// TwinCAT 3 PLC project OSCAT
// Title: OSCAT
// Company: RWTH Aachen University - E.ON Energy Research Center
// ProjectVersion: 1.1.2
// Description: This library is based on the OSCAT library (http://www.oscat.de/)
// ProgramVersion: 3.1.4022.1
// libraries:
//   Tc2_Standard, * (Beckhoff Automation GmbH)
// project tree:
//   oscat_basic/Data types/ CALENDAR.TcDUT (not stored), COMPLEX.TcDUT, CONSTANTS_LANGUAGE.TcDUT (not stored), CONSTANTS_LOCATION.TcDUT, CONSTANTS_MATH.TcDUT, CONSTANTS_PHYS.TcDUT, CONSTANTS_SETUP.TcDUT, ESR_DATA.TcDUT (not stored), CONTROL_MODE.TcDUT, FRACTION.TcDUT, HOLIDAY_DATA.TcDUT (not stored), REAL2.TcDUT, SDT.TcDUT, CONTROL_PARAMETERS.TcDUT, IO_TERMINAL_PARAMETERS.TcDUT, TIMER_EVENT.TcDUT (not stored), VECTOR_3.TcDUT
//   oscat_basic/Global Variables/ Constants_2.TcGVL, Globale_Variablen_2.TcGVL (not stored)
//   oscat_basic/POUs/Buffer Management/ BUFFER_COMP.TcPOU (not stored), BUFFER_SEARCH.TcPOU, BUFFER_TO_STRING.TcPOU, _BUFFER_INSERT.TcPOU, _BUFFER_UPPERCASE.TcPOU, _STRING_TO_BUFFER.TcPOU (not stored)
//   oscat_basic/POUs/Engineering/automation/ DRIVER_1.TcPOU, DRIVER_4.TcPOU (not stored), DRIVER_4C.TcPOU (not stored), FLOW_CONTROL.TcPOU, FT_Profile.TcPOU (not stored), INC_DEC.TcPOU (not stored), INTERLOCK.TcPOU, INTERLOCK_4.TcPOU, MANUAL.TcPOU, MANUAL_1.TcPOU, MANUAL_2.TcPOU (not stored), MANUAL_4.TcPOU (not stored), PARSET.TcPOU (not stored), PARSET2.TcPOU, SIGNAL.TcPOU (not stored), SIGNAL_4.TcPOU, SRAMP.TcPOU (not stored), TUNE.TcPOU (not stored), TUNE2.TcPOU (not stored)
//   oscat_basic/POUs/Engineering/Control/ BAND_B.TcPOU (not stored), CONTROL_SET1.TcPOU, CONTROL_SET2.TcPOU, CTRL_IN.TcPOU, CTRL_OUT.TcPOU, CTRL_PI.TcPOU, CTRL_PID.TcPOU, CTRL_PWM.TcPOU (not stored), DEAD_BAND.TcPOU (not stored), DEAD_BAND_A.TcPOU, DEAD_ZONE.TcPOU (not stored), DEAD_ZONE2.TcPOU (not stored), VOLTAGE_CONTROL.TcPOU, FB_CONTROL.TcPOU, FB_Integrate.TcPOU, FB_PID.TcPOU, FT_DERIV.TcPOU (not stored), FT_IMP.TcPOU, FT_INT.TcPOU (not stored), FT_INT2.TcPOU (not stored), FT_PD.TcPOU (not stored), FT_PDT1.TcPOU (not stored), FT_PI.TcPOU, FT_PID.TcPOU, FT_PIDW.TcPOU (not stored), FT_PIDWL.TcPOU, FT_PIW.TcPOU, FT_PIWL.TcPOU (not stored), FT_PT1.TcPOU, FT_PT2.TcPOU (not stored), FT_TN16.TcPOU, FT_TN64.TcPOU, FT_TN8.TcPOU, HYST.TcPOU, HYST_1.TcPOU, HYST_2.TcPOU, HYST_3.TcPOU, INTEGRATE.TcPOU (not stored)
//   oscat_basic/POUs/Engineering/Conversion/ ASTRO.TcPOU (not stored), BFT_TO_MS.TcPOU (not stored), C_TO_F.TcPOU, C_TO_K.TcPOU, DEG_TO_DIR.TcPOU, DIR_TO_DEG.TcPOU (not stored), ENERGY.TcPOU, F_TO_C.TcPOU (not stored), F_TO_OM.TcPOU (not stored), F_TO_PT.TcPOU, GEO_TO_DEG.TcPOU (not stored), KMH_TO_MS.TcPOU, K_TO_C.TcPOU (not stored), LENGTH.TcPOU (not stored), MS_TO_BFT.TcPOU (not stored), MS_TO_KMH.TcPOU, OM_TO_F.TcPOU (not stored), PRESSURE.TcPOU (not stored), PT_TO_F.TcPOU (not stored), SPEED.TcPOU (not stored), TEMPERATURE.TcPOU (not stored)
//   oscat_basic/POUs/Engineering/measurements/ ALARM_2.TcPOU (not stored), BAR_GRAPH.TcPOU (not stored), CALIBRATE.TcPOU, CYCLE_TIME.TcPOU (not stored), DT_SIMU.TcPOU (not stored), FLOW_METER.TcPOU, METER.TcPOU (not stored), METER_STAT.TcPOU, M_D.TcPOU, M_T.TcPOU (not stored), M_TX.TcPOU (not stored), ONTIME.TcPOU (not stored), TC_MS.TcPOU, TC_S.TcPOU (not stored), TC_US.TcPOU (not stored), T_PLC_MS.TcPOU (not stored), T_PLC_US.TcPOU
//   oscat_basic/POUs/Engineering/sensor/ MULTI_IN.TcPOU (not stored), RES_NI.TcPOU (not stored), RES_NTC.TcPOU, RES_PT.TcPOU, RES_SI.TcPOU (not stored), SENSOR_INT.TcPOU (not stored), TEMP_NI.TcPOU (not stored), TEMP_NTC.TcPOU, TEMP_PT.TcPOU, TEMP_SI.TcPOU
//   oscat_basic/POUs/Engineering/signal generators/ GEN_PULSE.TcPOU, GEN_PW2.TcPOU, GEN_RDM.TcPOU (not stored), GEN_RDT.TcPOU (not stored), GEN_RMP.TcPOU (not stored), GEN_SIN.TcPOU (not stored), GEN_SQR.TcPOU, PWM_DC.TcPOU (not stored), PWM_PW.TcPOU (not stored), RMP_B.TcPOU, RMP_SOFT.TcPOU, RMP_W.TcPOU, _RMP_B.TcPOU, _RMP_NEXT.TcPOU (not stored), _RMP_W.TcPOU (not stored)
//   oscat_basic/POUs/Engineering/signal processing/ AIN.TcPOU (not stored), AIN1.TcPOU, AOUT.TcPOU, AOUT1.TcPOU, BYTE_TO_RANGE.TcPOU, DELAY.TcPOU, DELAY_200.TcPOU, DELAY_4.TcPOU (not stored), FADE.TcPOU, FB_InLinear.TcPOU, FB_InOnOff.TcPOU, FB_OutLinear.TcPOU, FB_OutOnOff.TcPOU, FILTER_DW.TcPOU, FILTER_I.TcPOU, FILTER_MAV_DW.TcPOU (not stored), FILTER_MAV_W.TcPOU, FILTER_W.TcPOU (not stored), FILTER_WAV.TcPOU (not stored), MIX.TcPOU (not stored), MUX_R2.TcPOU (not stored), MUX_R4.TcPOU (not stored), OFFSET.TcPOU (not stored), OFFSET2.TcPOU (not stored), OVERRIDE.TcPOU, RANGE_TO_BYTE.TcPOU, RANGE_TO_WORD.TcPOU, SCALE.TcPOU (not stored), SCALE_B.TcPOU, SCALE_B2.TcPOU, SCALE_B4.TcPOU, SCALE_B8.TcPOU (not stored), SCALE_D.TcPOU, SCALE_R.TcPOU, SCALE_X2.TcPOU (not stored), SCALE_X4.TcPOU (not stored), SCALE_X8.TcPOU (not stored), SEL2_OF_3.TcPOU, SEL2_OF_3B.TcPOU (not stored), SH.TcPOU (not stored), SH_1.TcPOU, SH_2.TcPOU, SH_T.TcPOU, STAIR.TcPOU (not stored), STAIR2.TcPOU (not stored), TREND.TcPOU, TREND_DW.TcPOU (not stored), WORD_TO_RANGE.TcPOU
//   oscat_basic/POUs/List Processing/ LIST_ADD.TcPOU (not stored), LIST_CLEAN.TcPOU (not stored), LIST_GET.TcPOU, LIST_INSERT.TcPOU (not stored), LIST_LEN.TcPOU, LIST_NEXT.TcPOU, LIST_RETRIEVE.TcPOU (not stored), LIST_RETRIEVE_LAST.TcPOU (not stored)
//   oscat_basic/POUs/Logic/FF edge triggered/ COUNT_BR.TcPOU, COUNT_DR.TcPOU (not stored), FF_D2E.TcPOU, FF_D4E.TcPOU (not stored), FF_DRE.TcPOU, FF_JKE.TcPOU, FF_RSE.TcPOU (not stored), SELECT_8.TcPOU, SHR_4E.TcPOU (not stored), SHR_4UDE.TcPOU, SHR_8PLE.TcPOU (not stored), SHR_8UDE.TcPOU, TOGGLE.TcPOU (not stored)
//   oscat_basic/POUs/Logic/FF pulse triggered/ LTCH.TcPOU (not stored), LTCH_4.TcPOU (not stored), STORE_8.TcPOU
//   oscat_basic/POUs/Logic/gate logic/ BCDC_TO_INT.TcPOU, BIT_COUNT.TcPOU, BIT_LOAD_B.TcPOU, BIT_LOAD_B2.TcPOU, BIT_LOAD_DW.TcPOU, BIT_LOAD_DW2.TcPOU (not stored), BIT_LOAD_W.TcPOU (not stored), BIT_LOAD_W2.TcPOU, BIT_OF_DWORD.TcPOU (not stored), BIT_TOGGLE_B.TcPOU (not stored), BIT_TOGGLE_DW.TcPOU, BIT_TOGGLE_W.TcPOU, BYTE_OF_BIT.TcPOU (not stored), BYTE_OF_DWORD.TcPOU, BYTE_TO_BITS.TcPOU (not stored), BYTE_TO_GRAY.TcPOU, CHECK_PARITY.TcPOU (not stored), CHK_REAL.TcPOU, DEC_2.TcPOU, DEC_4.TcPOU, DEC_8.TcPOU (not stored), DWORD_OF_BYTE.TcPOU (not stored), DWORD_OF_WORD.TcPOU, DW_TO_REAL.TcPOU, GRAY_TO_BYTE.TcPOU, INT_TO_BCDC.TcPOU (not stored), MUX_2.TcPOU, MUX_4.TcPOU, PARITY.TcPOU, REAL_TO_DW.TcPOU, REFLECT.TcPOU, REVERSE.TcPOU (not stored), SHL1.TcPOU, SHR1.TcPOU (not stored), SWAP_BYTE.TcPOU (not stored), SWAP_BYTE2.TcPOU (not stored), WORD_OF_BYTE.TcPOU (not stored), WORD_OF_DWORD.TcPOU
//   oscat_basic/POUs/Logic/generators/ A_TRIG.TcPOU (not stored), B_TRIG.TcPOU, CLICK_CNT.TcPOU, CLICK_DEC.TcPOU (not stored), CLK_DIV.TcPOU (not stored), CLK_N.TcPOU (not stored), CLK_PRG.TcPOU, CLK_PULSE.TcPOU, CYCLE_4.TcPOU (not stored), D_TRIG.TcPOU, GEN_BIT.TcPOU (not stored), GEN_SQ.TcPOU, SCHEDULER.TcPOU (not stored), SCHEDULER_2.TcPOU (not stored), SEQUENCE_4.TcPOU (not stored), SEQUENCE_64.TcPOU, SEQUENCE_8.TcPOU, TMAX.TcPOU, TMIN.TcPOU, TOF_1.TcPOU (not stored), TONOF.TcPOU, TP_1.TcPOU (not stored), TP_1D.TcPOU (not stored), TP_X.TcPOU
//   oscat_basic/POUs/Logic/memory/ FIFO_16.TcPOU (not stored), FIFO_32.TcPOU, STACK_16.TcPOU, STACK_32.TcPOU
//   oscat_basic/POUs/Logic/Others/ CRC_GEN.TcPOU (not stored), MATRIX.TcPOU (not stored), PIN_CODE.TcPOU
//   oscat_basic/POUs/Mathematical/ ACOSH.TcPOU, ACOTH.TcPOU (not stored), AGDF.TcPOU (not stored), ASINH.TcPOU, ATAN2.TcPOU (not stored), ATANH.TcPOU (not stored), BETA.TcPOU, BINOM.TcPOU, CAUCHY.TcPOU, CAUCHYCD.TcPOU (not stored), CEIL.TcPOU (not stored), CEIL2.TcPOU (not stored), CMP.TcPOU, COSH.TcPOU, COTH.TcPOU, DEC1.TcPOU, DEG.TcPOU (not stored), DIFFER.TcPOU (not stored), D_TRUNC.TcPOU, ERF.TcPOU, ERFC.TcPOU, EVEN.TcPOU, EXP10.TcPOU, EXPN.TcPOU (not stored), FACT.TcPOU (not stored), FIB.TcPOU, FLOOR.TcPOU (not stored), FLOOR2.TcPOU, FRACT.TcPOU (not stored), GAMMA.TcPOU, GAUSS.TcPOU, GAUSSCD.TcPOU, GCD.TcPOU (not stored), GDF.TcPOU, GOLD.TcPOU, HYPOT.TcPOU, INC.TcPOU (not stored), INC1.TcPOU, INC2.TcPOU (not stored), INV.TcPOU (not stored), LAMBERT_W.TcPOU (not stored), LANGEVIN.TcPOU, MAX3.TcPOU, MID3.TcPOU, MIN3.TcPOU (not stored), MODR.TcPOU, MUL_ADD.TcPOU, NEGX.TcPOU, RAD.TcPOU (not stored), RDM.TcPOU (not stored), RDM2.TcPOU, RDMDW.TcPOU, REAL_TO_FRAC.TcPOU, RND.TcPOU (not stored), ROUND.TcPOU (not stored), SGN.TcPOU, SIGMOID.TcPOU, SIGN_I.TcPOU (not stored), SIGN_R.TcPOU (not stored), SINC.TcPOU, SINH.TcPOU (not stored), SQRTN.TcPOU, TANC.TcPOU, TANH.TcPOU, WINDOW.TcPOU, WINDOW2.TcPOU
//   oscat_basic/POUs/Mathematical/Array/ ARRAY_AVG.TcPOU (not stored), ARRAY_GAV.TcPOU, ARRAY_HAV.TcPOU, ARRAY_MAX.TcPOU, ARRAY_MIN.TcPOU (not stored), ARRAY_SDV.TcPOU (not stored), ARRAY_SPR.TcPOU, ARRAY_SUM.TcPOU, ARRAY_TREND.TcPOU (not stored), ARRAY_VAR.TcPOU (not stored), IS_SORTED.TcPOU (not stored), _ARRAY_ABS.TcPOU (not stored), _ARRAY_ADD.TcPOU (not stored), _ARRAY_INIT.TcPOU (not stored), _ARRAY_MEDIAN.TcPOU (not stored), _ARRAY_MUL.TcPOU (not stored), _ARRAY_SHUFFLE.TcPOU (not stored), _ARRAY_SORT.TcPOU (not stored)
//   oscat_basic/POUs/Mathematical/Complex/ CABS.TcPOU (not stored), CACOS.TcPOU (not stored), CACOSH.TcPOU (not stored), CADD.TcPOU (not stored), CARG.TcPOU (not stored), CASIN.TcPOU (not stored), CASINH.TcPOU (not stored), CATAN.TcPOU (not stored), CATANH.TcPOU (not stored), CCON.TcPOU (not stored), CCOS.TcPOU (not stored), CCOSH.TcPOU (not stored), CDIV.TcPOU (not stored), CEXP.TcPOU (not stored), CINV.TcPOU (not stored), CLOG.TcPOU (not stored), CMUL.TcPOU (not stored), CPOL.TcPOU (not stored), CPOW.TcPOU (not stored), CSET.TcPOU (not stored), CSIN.TcPOU (not stored), CSINH.TcPOU (not stored), CSQRT.TcPOU (not stored), CSUB.TcPOU (not stored), CTAN.TcPOU (not stored), CTANH.TcPOU (not stored)
//   oscat_basic/POUs/Mathematical/Double Precision/ R2_ABS.TcPOU (not stored), R2_ADD.TcPOU (not stored), R2_ADD2.TcPOU (not stored), R2_MUL.TcPOU (not stored), R2_SET.TcPOU (not stored)
//   oscat_basic/POUs/Mathematical/functions/ FRMP_B.TcPOU (not stored), FT_AVG.TcPOU (not stored), FT_AVG_200.TcPOU (not stored), FT_MIN_MAX.TcPOU (not stored), FT_RMP.TcPOU (not stored), F_LIN.TcPOU (not stored), F_LIN2.TcPOU (not stored), F_POLY.TcPOU (not stored), F_POWER.TcPOU (not stored), F_QUAD.TcPOU (not stored), LINEAR_INT.TcPOU (not stored), POLYNOM_INT.TcPOU (not stored)
//   oscat_basic/POUs/Mathematical/Geometry/ CIRCLE_A.TcPOU (not stored), CIRCLE_C.TcPOU (not stored), CIRCLE_SEG.TcPOU (not stored), CONE_V.TcPOU (not stored), ELLIPSE_A.TcPOU (not stored), ELLIPSE_C.TcPOU (not stored), SPHERE_V.TcPOU (not stored), TRIANGLE_A.TcPOU (not stored)
//   oscat_basic/POUs/Mathematical/Vektormathematik/ V3_ABS.TcPOU (not stored), V3_ADD.TcPOU (not stored), V3_ANG.TcPOU (not stored), V3_DPRO.TcPOU (not stored), V3_NORM.TcPOU (not stored), V3_NUL.TcPOU (not stored), V3_PAR.TcPOU (not stored), V3_REV.TcPOU (not stored), V3_SMUL.TcPOU (not stored), V3_SUB.TcPOU (not stored), V3_XANG.TcPOU (not stored), V3_XPRO.TcPOU (not stored), V3_YANG.TcPOU (not stored), V3_ZANG.TcPOU (not stored)
//   oscat_basic/POUs/Other/ ESR_COLLECT.TcPOU, ESR_MON_B8.TcPOU (not stored), ESR_MON_R4.TcPOU, ESR_MON_X8.TcPOU (not stored), OSCAT_VERSION.TcPOU (not stored), STATUS_TO_ESR.TcPOU
//   oscat_basic/POUs/String/ BIN_TO_BYTE.TcPOU (not stored), BIN_TO_DWORD.TcPOU, BYTE_TO_STRB.TcPOU (not stored), BYTE_TO_STRH.TcPOU, CAPITALIZE.TcPOU, CHARCODE.TcPOU, CHARNAME.TcPOU, CHR_TO_STRING.TcPOU (not stored), CLEAN.TcPOU (not stored), CODE.TcPOU (not stored), COUNT_CHAR.TcPOU (not stored), COUNT_SUBSTRING.TcPOU (not stored), DEC_TO_BYTE.TcPOU (not stored), DEC_TO_DWORD.TcPOU, DEC_TO_INT.TcPOU (not stored), DEL_CHARS.TcPOU (not stored), DT_TO_STRF.TcPOU (not stored), DWORD_TO_STRB.TcPOU, DWORD_TO_STRF.TcPOU (not stored), DWORD_TO_STRH.TcPOU (not stored), EXEC.TcPOU (not stored), FILL.TcPOU (not stored), FINDB.TcPOU (not stored), FINDB_NONUM.TcPOU, FINDB_NUM.TcPOU (not stored), FINDP.TcPOU, FIND_CHAR.TcPOU, FIND_CTRL.TcPOU, FIND_NONUM.TcPOU (not stored), FIND_NUM.TcPOU (not stored), FIX.TcPOU, FLOAT_TO_REAL.TcPOU, FSTRING_TO_BYTE.TcPOU (not stored), FSTRING_TO_DT.TcPOU, FSTRING_TO_DWORD.TcPOU, FSTRING_TO_MONTH.TcPOU, FSTRING_TO_WEEK.TcPOU (not stored), FSTRING_TO_WEEKDAY.TcPOU (not stored), HEX_TO_BYTE.TcPOU, HEX_TO_DWORD.TcPOU, ISC_ALPHA.TcPOU, ISC_CTRL.TcPOU (not stored), ISC_HEX.TcPOU, ISC_LOWER.TcPOU (not stored), ISC_NUM.TcPOU (not stored), ISC_UPPER.TcPOU, IS_ALNUM.TcPOU, IS_ALPHA.TcPOU (not stored), IS_CC.TcPOU, IS_CTRL.TcPOU (not stored), IS_HEX.TcPOU, IS_LOWER.TcPOU, IS_NCC.TcPOU (not stored), IS_NUM.TcPOU, IS_UPPER.TcPOU (not stored), LOWERCASE.TcPOU (not stored), MESSAGE_4R.TcPOU, MESSAGE_8.TcPOU (not stored), MIRROR.TcPOU, MONTH_TO_STRING.TcPOU, OCT_TO_BYTE.TcPOU, OCT_TO_DWORD.TcPOU (not stored), REAL_TO_STRF.TcPOU, REPLACE_ALL.TcPOU (not stored), REPLACE_CHARS.TcPOU, REPLACE_UML.TcPOU, TICKER.TcPOU, TO_LOWER.TcPOU (not stored), TO_UML.TcPOU, TO_UPPER.TcPOU (not stored), TRIM.TcPOU, TRIM1.TcPOU (not stored), TRIME.TcPOU, UPPERCASE.TcPOU, WEEKDAY_TO_STRING.TcPOU
//   oscat_basic/POUs/Time&Date/ CALENDAR_CALC.TcPOU (not stored), DATE_ADD.TcPOU, DAYS_DELTA.TcPOU, DAYS_IN_MONTH.TcPOU, DAYS_IN_YEAR.TcPOU (not stored), DAY_OF_DATE.TcPOU (not stored), DAY_OF_MONTH.TcPOU, DAY_OF_WEEK.TcPOU (not stored), DAY_OF_YEAR.TcPOU, DAY_TO_TIME.TcPOU (not stored), DCF77.TcPOU (not stored), DST.TcPOU, DT2_TO_SDT.TcPOU (not stored), DT_TO_SDT.TcPOU, EASTER.TcPOU (not stored), EVENTS.TcPOU (not stored), HOLIDAY.TcPOU, HOUR.TcPOU (not stored), HOUR_OF_DT.TcPOU (not stored), HOUR_TO_TIME.TcPOU, HOUR_TO_TOD.TcPOU (not stored), JD2000.TcPOU (not stored), LEAP_DAY.TcPOU, LEAP_OF_DATE.TcPOU (not stored), LEAP_YEAR.TcPOU (not stored), LTIME_TO_UTC.TcPOU, MINUTE.TcPOU (not stored), MINUTE_OF_DT.TcPOU, MINUTE_TO_TIME.TcPOU, MONTH_BEGIN.TcPOU, MONTH_END.TcPOU (not stored), MONTH_OF_DATE.TcPOU, MULTIME.TcPOU, PERIOD.TcPOU, PERIOD2.TcPOU, REFRACTION.TcPOU, RTC_2.TcPOU, RTC_MS.TcPOU, SDT_TO_DATE.TcPOU, SDT_TO_DT.TcPOU (not stored), SDT_TO_TOD.TcPOU, SECOND.TcPOU, SECOND_OF_DT.TcPOU (not stored), SECOND_TO_TIME.TcPOU, SET_DATE.TcPOU (not stored), SET_DT.TcPOU, SET_TOD.TcPOU, SUN_MIDDAY.TcPOU, SUN_POS.TcPOU, SUN_TIME.TcPOU, TIMECHECK.TcPOU, TON_P.TcPOU, UTC_TO_LTIME.TcPOU (not stored), WORK_WEEK.TcPOU (not stored), YEAR_BEGIN.TcPOU (not stored), YEAR_END.TcPOU, YEAR_OF_DATE.TcPOU
//   oscat_building/Global Variables/ Constants.TcGVL, Globale_Variablen.TcGVL (not stored), Setup_Data.TcGVL
//   oscat_building/POUs/actuators/ ACTUATOR_2P.TcPOU (not stored), ACTUATOR_3P.TcPOU (not stored), ACTUATOR_A.TcPOU (not stored), ACTUATOR_COIL.TcPOU (not stored), ACTUATOR_PUMP.TcPOU (not stored), ACTUATOR_UD.TcPOU, AUTORUN.TcPOU
//   oscat_building/POUs/electrical/ CLICK.TcPOU, CLICK_MODE.TcPOU, DEBOUNCE.TcPOU (not stored), DIMM_2.TcPOU (not stored), DIMM_I.TcPOU (not stored), F_LAMP.TcPOU, PULSE_LENGTH.TcPOU, PULSE_T.TcPOU (not stored), SWITCH_I.TcPOU, SWITCH_X.TcPOU (not stored), SW_RECONFIG.TcPOU (not stored), TIMER_1.TcPOU (not stored), TIMER_2.TcPOU, TIMER_EVENT_DECODE.TcPOU (not stored), TIMER_EXT.TcPOU, TIMER_P4.TcPOU
//   oscat_building/POUs/HLK/ AIR_DENSITY.TcPOU (not stored), AIR_ENTHALPY.TcPOU, BOILER.TcPOU, BURNER.TcPOU (not stored), DEW_CON.TcPOU (not stored), DEW_RH.TcPOU, DEW_TEMP.TcPOU (not stored), HEAT_INDEX.TcPOU, HEAT_METER.TcPOU (not stored), HEAT_TEMP.TcPOU, LEGIONELLA.TcPOU (not stored), SDD.TcPOU (not stored), SDD_NH3.TcPOU (not stored), SDT_NH3.TcPOU (not stored), TANK_LEVEL.TcPOU (not stored), TANK_VOL1.TcPOU (not stored), TANK_VOL2.TcPOU, TEMP_EXT.TcPOU (not stored), T_AVG24.TcPOU, WATER_CP.TcPOU, WATER_DENSITY.TcPOU (not stored), WATER_ENTHALPY.TcPOU, WCT.TcPOU
//   oscat_building/POUs/Jalousie/ BLIND_ACTUATOR.TcPOU (not stored), BLIND_CONTROL.TcPOU (not stored), BLIND_CONTROL_S.TcPOU, BLIND_INPUT.TcPOU, BLIND_NIGHT.TcPOU, BLIND_SCENE.TcPOU, BLIND_SECURITY.TcPOU, BLIND_SET.TcPOU (not stored), BLIND_SHADE.TcPOU, BLIND_SHADE_S.TcPOU (not stored)
//   oscat_building/POUs/Other/ BUILDING_VERSION.TcPOU
//   oscat_network/Data types/DATA_LOG/ DLOG_DATA.TcDUT, LOG_CONTROL.TcDUT, MYSQL_COM.TcDUT, PRINTF_DATA.TcDUT, UNI_CIRCULAR_BUFFER_DATA.TcDUT, us_LOG_VIEWPORT.TcDUT
//   oscat_network/Data types/FILE_SERVER/ FILE_PATH_DATA.TcDUT, FILE_SERVER_DATA.TcDUT
//   oscat_network/Data types/NETWORK/ IP2GEO_DATA.TcDUT, IP_C.TcDUT, IP_FIFO_DATA.TcDUT, NETWORK_BUFFER.TcDUT, NETWORK_BUFFER_SHORT.TcDUT, NW_BUF_LONG.TcDUT, NW_BUF_SHORT.TcDUT, URL.TcDUT, VMAP_DATA.TcDUT, XML_CONTROL.TcDUT
//   oscat_network/Data types/NET_VAR/ NET_VAR_DATA.TcDUT
//   oscat_network/Data types/TELNET_VISION/ us_TN_INPUT_CONTROL.TcDUT, us_TN_INPUT_CONTROL_DATA.TcDUT, us_TN_MENU.TcDUT, us_TN_MENU_POPUP.TcDUT, us_TN_SCREEN.TcDUT
//   oscat_network/Data types/WEATHER/ WORLD_WEATHER_CUR.TcDUT, WORLD_WEATHER_DATA.TcDUT, WORLD_WEATHER_DAY.TcDUT, YAHOO_WEATHER_DATA.TcDUT
//   oscat_network/Global Variables/ Constants_1.TcGVL, Globale_Variablen_1.TcGVL
//   oscat_network/POUs/CO_NVERT/ BASE64_DECODE_STREAM_1.TcPOU, BASE64_DECODE_STR_1.TcPOU, BASE64_ENCODE_STREAM_1.TcPOU, BASE64_ENCODE_STR_1.TcPOU, HTML_DECODE_1.TcPOU, HTML_ENCODE_1.TcPOU, IP4_CHECK_1.TcPOU, IP4_DECODE_1.TcPOU, IP4_TO_STRING_1.TcPOU, IS_IP4_1.TcPOU, IS_URLCHR_1.TcPOU, MD5_AUX_1.TcPOU, MD5_CRAM_AUTH_1.TcPOU, MD5_STREAM_1.TcPOU, MD5_STR_1.TcPOU, MD5_TO_STRH_1.TcPOU, RC4_CRYPT_STREAM_1.TcPOU, SHA1_STREAM_1.TcPOU, SHA1_STR_1.TcPOU, SHA1_TO_STRH_1.TcPOU, STRING_TO_URL_1.TcPOU, URL_DECODE_1.TcPOU, URL_ENCODE_1.TcPOU, URL_TO_STRING_1.TcPOU
//   oscat_network/POUs/DATA_LOG/ DLOG_BOOL_1.TcPOU, DLOG_DINT_1.TcPOU, DLOG_DT_1.TcPOU, DLOG_FILE_TO_FTP_1.TcPOU, DLOG_FILE_TO_SMTP_1.TcPOU, DLOG_REAL_1.TcPOU, DLOG_STORE_FILE_CSV_1.TcPOU, DLOG_STORE_FILE_HTML_1.TcPOU, DLOG_STORE_FILE_XML_1.TcPOU, DLOG_STORE_RRD_1.TcPOU, DLOG_STRING_1.TcPOU, UNI_CIRCULAR_BUFFER_1.TcPOU
//   oscat_network/POUs/DEMO/ BASE64_DEMO_1.TcPOU, CSV_PARSER_BUF_DEMO_1.TcPOU, CSV_PARSER_FILE_DEMO_1.TcPOU, DLOG_FILE_CSV_DEMO_1.TcPOU, DLOG_FILE_CSV_FTP_DEMO_1.TcPOU, DLOG_FILE_CSV_SMTP_DEMO_1.TcPOU, DLOG_FILE_HTML_DEMO_1.TcPOU, DLOG_FILE_XML_DEMO_1.TcPOU, DLOG_RRD_DEMO_1.TcPOU, DNS_DYN_DEMO_1.TcPOU, DNS_REV_DEMO_1.TcPOU, DNS_SNTP_SYSLOG_DEMO_1.TcPOU, FILE_BLOCK_DEMO_1.TcPOU, FTP_CLIENT_DEMO_1.TcPOU, GET_WAN_IP_DEMO_1.TcPOU, HTTP_DEMO_1.TcPOU, INI_PARSER_BUF_DEMO_1.TcPOU, INI_PARSER_FILE_DEMO_1.TcPOU, IP2GEO_DEMO_1.TcPOU, IRTRANS_DEMO_1.TcPOU, MB_CLIENT_DEMO_1.TcPOU, MB_SERVER_DEMO_1.TcPOU, MD5_CRAM_AUTH_DEMO_1.TcPOU, NET_VAR_MASTER_DEMO_1.TcPOU, NET_VAR_SLAVE_DEMO_1.TcPOU, RC4_CRYPT_DEMO_1.TcPOU, SHA1_MD5_DEMO_1.TcPOU, SMTP_CLIENT_DEMO_1.TcPOU, SPIDER_DEMO_1.TcPOU, TELNET_LOG_DEMO_1.TcPOU, TELNET_PRINT_DEMO_1.TcPOU, TN_VISION_DEMO_1_1.TcPOU, TN_VISION_DEMO_2_1.TcPOU, WORLD_WEATHER_DEMO_1.TcPOU, YAHOO_WEATHER_DEMO_1.TcPOU
//   oscat_network/POUs/DRIVER/ IRTRANS_DECODE_1.TcPOU, IRTRANS_RCV_1_1.TcPOU, IRTRANS_RCV_4_1.TcPOU, IRTRANS_RCV_8_1.TcPOU, IRTRANS_SERVER_1.TcPOU, IRTRANS_SND_1_1.TcPOU, IRTRANS_SND_4_1.TcPOU, IRTRANS_SND_8_1.TcPOU
//   oscat_network/POUs/FILE/ CSV_PARSER_BUF_1.TcPOU, CSV_PARSER_FILE_1.TcPOU, FILE_BLOCK_1.TcPOU, FILE_PATH_SPLIT_1.TcPOU, INI_PARSER_BUF_1.TcPOU, INI_PARSER_FILE_1.TcPOU
//   oscat_network/POUs/HARDWARE/ FILE_SERVER_1.TcPOU, IP_CONTROL2_1.TcPOU, IP_CONTROL_1.TcPOU, IP_CONTROL_RESET_1.TcPOU
//   oscat_network/POUs/NETWORK/ DNS_CLIENT.TcPOU, DNS_DYN.TcPOU, DNS_REV_CLIENT.TcPOU, FTP_CLIENT.TcPOU, GET_WAN_IP.TcPOU, HTTP_GET.TcPOU, IP2GEO.TcPOU, IP_FIFO.TcPOU, LOG_MSG.TcPOU, LOG_VIEWPORT.TcPOU, MB_CLIENT.TcPOU, MB_SERVER.TcPOU, MB_VMAP.TcPOU, PRINT_SF.TcPOU, READ_HTTP.TcPOU, SMTP_CLIENT.TcPOU, SNTP_CLIENT.TcPOU, SNTP_SERVER.TcPOU, SPIDER_ACCESS.TcPOU, SYS_LOG.TcPOU, TELNET_LOG.TcPOU, TELNET_PRINT.TcPOU, XML_READER.TcPOU
//   oscat_network/POUs/NET_VAR/ NET_VAR_BOOL8.TcPOU, NET_VAR_BUFFER.TcPOU, NET_VAR_CONTROL.TcPOU, NET_VAR_DWORD8.TcPOU, NET_VAR_REAL8.TcPOU, NET_VAR_STRING.TcPOU, NET_VAR_X8.TcPOU
//   oscat_network/POUs/OTHER/ ELEMENT_COUNT.TcPOU, ELEMENT_GET.TcPOU, NETWORK_VERSION.TcPOU
//   oscat_network/POUs/TELNET_VISION/ TN_FRAMEWORK.TcPOU, TN_INPUT_CONTROL.TcPOU, TN_INPUT_EDIT_LINE.TcPOU, TN_INPUT_MENU_BAR.TcPOU, TN_INPUT_MENU_POPUP.TcPOU, TN_INPUT_SELECT_POPUP.TcPOU, TN_INPUT_SELECT_TEXT.TcPOU, TN_RECEIVE.TcPOU, TN_SC_ADD_SHADOW.TcPOU, TN_SC_AREA_RESTORE.TcPOU, TN_SC_AREA_SAVE.TcPOU, TN_SC_BOX.TcPOU, TN_SC_FILL.TcPOU, TN_SC_LINE.TcPOU, TN_SC_READ_ATTR.TcPOU, TN_SC_READ_CHAR.TcPOU, TN_SC_SHADOW_ATTR.TcPOU, TN_SC_VIEWPORT.TcPOU, TN_SC_WRITE.TcPOU, TN_SC_WRITE_ATTR.TcPOU, TN_SC_WRITE_C.TcPOU, TN_SC_WRITE_CHAR.TcPOU, TN_SC_WRITE_EOS.TcPOU, TN_SC_XY2_ERROR.TcPOU, TN_SC_XY_ERROR.TcPOU, TN_SEND_ROWS.TcPOU
//   oscat_network/POUs/WEATHER/ MOON_PHASE.TcPOU, WORLD_WEATHER.TcPOU, WORLD_WEATHER_DESC_GE.TcPOU, WORLD_WEATHER_ICON_OSCAT.TcPOU, YAHOO_WEATHER.TcPOU, YAHOO_WEATHER_DESC_GE.TcPOU, YAHOO_WEATHER_ICON_OSCAT.TcPOU

// ---- oscat_basic/Data types/COMPLEX.TcDUT
TYPE COMPLEX :
STRUCT
	re : REAL;
	im : REAL;
END_STRUCT
END_TYPE

// ---- oscat_basic/Data types/CONSTANTS_LOCATION.TcDUT
TYPE CONSTANTS_LOCATION :
STRUCT
	(* location setup *)
	DEFAULT : INT := 1; (* 1=germany, 2=austria 3=france 4=belgium-german 5= italien-Südtirol *)
	LMAX : INT := 5;

	(* language spoken in the location *)
	LANGUAGE : ARRAY[1..5] OF INT :=[ 2, 2, 3, 2, 2];

END_STRUCT
END_TYPE

// ---- oscat_basic/Data types/CONSTANTS_MATH.TcDUT
TYPE CONSTANTS_MATH :
STRUCT
	PI : REAL := 	3.14159265358979323846264338327950288;		(* Kreiszahl PI *)
	PI2 : REAL := 	6.28318530717958647692528676655900576;	(* PI * 2 *)
	PI4 : REAL :=  12.56637061435917295385057353311801152;	(* PI * 4 *)
	PI05 : REAL :=  1.5707963267949;							(* PI / 2 *)
	PI025 : REAL := 0.785398163397448;							(* PI / 4 *)
	PI_INV : REAL := 0.318309886183791;						(* 1 / PI *)
	E : REAL := 	2.71828182845904523536028747135266249;		(* Euler constant e *)
	E_INV : REAL := 0.367879441171442;							(* 1 / e *)
	SQ2 : REAL :=	1.4142135623731;							(* Wurzel von 2 *)
	FACTS : ARRAY[0..12] OF DINT :=[ 1,1,2,6,24,120,720,5040,40320,362880,3628800,39916800,479001600];
END_STRUCT
END_TYPE

// ---- oscat_basic/Data types/CONSTANTS_PHYS.TcDUT
TYPE CONSTANTS_PHYS :
STRUCT
	C : REAL := 299792458.0;				(* Lichtgeschwindigkeit in m/s *)
	E : REAL := 1.60217653E-19;				(* elementarladung in Colomb = A * s *)
	G : REAL := 9.80665; 						(* Erdbeschleunigung in m / s² *)
	T0 : REAL := -273.15;						(* absoluter Nullpunkt in °C *)
	RU : REAL := 8.314472; 					(* Universelle Gaskonstante in J / (mol · K) *)
	PN : REAL := 101325.0;					(* NormalDruck in Pa *)
END_STRUCT
END_TYPE

// ---- oscat_basic/Data types/CONSTANTS_SETUP.TcDUT
TYPE CONSTANTS_SETUP :
STRUCT
	(* setup Parameters *)
	EXTENDED_ASCII : BOOL := TRUE;
	CHARNAMES : ARRAY[1..4] OF STRING(253) :=[ ';"&quot;&&amp;<&lt;>&gt;€&euro; &nbsp;¡&iexcl;¢&cent;£&pound;¤&curren;¥&yen;¦&brvbar;§&sect;¨&uml;©&copy;ª&ordf;«&laquo;¬&not;­&shy;®&reg;¯&macr;°&deg;±&plusmn;²&sup2;³&sup3;´&acute;µ&micro;¶&para;·&middot;¸&cedil;¹&sup1;º&ordm;»&raquo;¼&frac14;Û&Ucirc;',
		';¾&frac34;¿&iquest;À&Agrave;Á&Aacute;Â&Acirc;Ã&Atilde;Ä&Auml;Å&Aring;Æ&AElig;Ç&Ccedil;È&Egrave;É&Eacute;Ê&Ecirc;Ë&Euml;Ì&Igrave;Í&Iacute;Î&Icirc;Ï&Iuml;Ð&ETH;Ñ&Ntilde;Ò&Ograve;Ó&Oacute;Ô&Ocirc;Õ&Otilde;Ö&Ouml;×&times;Ø&Oslash;Ù&Ugrave;Ú&Uacute;½&frac12;',
		';Ü&Uuml;Ý&Yacute;Þ&THORN;ß&szlig;à&agrave;á&aacute;â&acirc;ã&atilde;ä&auml;å&aring;æ&aelig;ç&ccedil;è&egrave;é&eacute;ê&ecirc;ë&euml;ì&igrave;í&iacute;î&icirc;ï&iuml;ð&eth;ñ&ntilde;ò&ograve;ó&oacute;ô&ocirc;õ&otilde;ö&ouml;÷&divide;ø&oslash;ù&ugrave;',
		';ú&uacute;û&ucirc;ü&uuml;ý&yacute;þ&thorn;ÿ&yuml;'];
	MTH_OFS : ARRAY[1..12] OF INT :=[ 0,31,59,90,120,151,181,212,243,273,304,334];
	DECADES : ARRAY[0..8] OF REAL :=[ 1.0,10.0,100.0,1000.0,10000.0,10000.0,100000.0,1000000.0,10000000.0];
END_STRUCT
END_TYPE

// ---- oscat_basic/Data types/CONTROL_MODE.TcDUT
{attribute 'qualified_only'}
{attribute 'strict'}
TYPE CONTROL_MODE :
(
	Off,				(*0*)
	Manual,				(*1*)
	Auto				(*2*)
);
END_TYPE

// ---- oscat_basic/Data types/FRACTION.TcDUT
TYPE FRACTION :
STRUCT
	NUMERATOR : INT;
	DENOMINATOR : INT;
END_STRUCT
END_TYPE

// ---- oscat_basic/Data types/REAL2.TcDUT
TYPE REAL2 :
STRUCT
	R1 : REAL;	(* small value *)
	RX : REAL;	(* big value *)
END_STRUCT
END_TYPE

// ---- oscat_basic/Data types/SDT.TcDUT
TYPE SDT :
STRUCT
	YEAR : INT;
	MONTH : INT;
	DAY : INT;
	WEEKDAY : INT;
	HOUR : INT;
	MINUTE : INT;
	SECOND : INT;
	MS : INT;
END_STRUCT
END_TYPE

// ---- oscat_basic/Data types/CONTROL_PARAMETERS.TcDUT
TYPE CONTROL_PARAMETERS :
STRUCT
	Kp		:	REAL;	
	Ti		:	REAL;
	Td		:	REAL;
	LimLow	:	REAL;
	LimHigh	:	REAL;
	bReverseActing	:	BOOL;
	RST	:	BOOL;	//Reset
END_STRUCT
END_TYPE

// ---- oscat_basic/Data types/IO_TERMINAL_PARAMETERS.TcDUT
TYPE IO_TERMINAL_PARAMETERS :
STRUCT
	cValue1Raw 				: REAL;			//Maximaler Klemmenwert (z.B. 32767)
	cValue2Raw				: REAL;			//Minimaler Klemmenwert (z.B. 0)
	cValue1 				: REAL;			//Maximaler Bildwert (z.B. 100%)
	cValue2 				: REAL;			//Minimaler Bildwert (z.B. 0%)
	cAVG_N					: INT;
END_STRUCT
END_TYPE

// ---- oscat_basic/Data types/VECTOR_3.TcDUT
TYPE VECTOR_3 :
STRUCT
	X : REAL;
	Y : REAL;
	Z : REAL;
END_STRUCT
END_TYPE

// ---- oscat_network/Data types/DATA_LOG/DLOG_DATA.TcDUT
TYPE DLOG_DATA :
STRUCT
	STORE_TYPE : BYTE;
	ADD_HEADER : BOOL;
	ADD_DATA : BOOL;
	ADD_DATA_REQ : BOOL;
	CLOCK_TRIG : BOOL;
	ID_MAX : USINT;
	DTI : DT;
	UCB : UNI_CIRCULAR_BUFFER_DATA;
	NEW_FILE : STRING;
	NEW_FILE_RTRIG : BOOL;
END_STRUCT
END_TYPE

// ---- oscat_network/Data types/DATA_LOG/LOG_CONTROL.TcDUT
TYPE LOG_CONTROL :
STRUCT
	NEW_MSG : STRING(LOG_SIZE); (* neue Nachricht für den Datenbuffer *)
	NEW_MSG_OPTION : DWORD;
	LEVEL : BYTE;
	SIZE : INT := LOG_MAX; (* Anzahl der Strings im LOG_DATA *)
	RESET : BOOL; (* Nachrichtenbuffer löschen *)
	PRINTF : PRINTF_DATA; (* Array PRINTF Parameter *)
	MSG : ARRAY [0..LOG_MAX] OF STRING(LOG_SIZE); (* Array Message *)
	MSG_OPTION : ARRAY [0..LOG_MAX] OF DWORD; (* Array Options *)
	UPDATE_COUNT : UINT; (* Updatezähler *)
	IDX : INT; (* aktueller Nachrichten-Index *)
	RING_MODE : BOOL; (* Bufferüberlauf erkannt *)
END_STRUCT
END_TYPE

// ---- oscat_network/Data types/DATA_LOG/MYSQL_COM.TcDUT
TYPE MYSQL_COM :
STRUCT
	SERVER_PROTOCOL_VERSION : BYTE;
	SERVER_CAPABILITIES : WORD;
	SERVER_STATUS : WORD;
	SERVER_LANGUAGE : BYTE;
	S_BUF : NETWORK_BUFFER;
	R_BUF : NETWORK_BUFFER;

	(* eingänge *)
	SQL_CON : BOOL;
	SQL_START : BOOL;
	SQL_URL : STRING(STRING_LENGTH);
	SQL_PACKET_NO : BYTE;

	TIMEOUT : TIME;
	DNS_IP4 : DWORD;

	(* ausgänge *)
	SQL_LOGGED_IN : BOOL;
	SQL_RCV_STATE : BYTE;
	SQL_ERROR : STRING(STRING_LENGTH);
	ERROR_C : DWORD;
	ERROR_T : BYTE;

END_STRUCT
END_TYPE

// ---- oscat_network/Data types/DATA_LOG/PRINTF_DATA.TcDUT
TYPE PRINTF_DATA : ARRAY [1..11]  OF STRING(LOG_SIZE);
END_TYPE

// ---- oscat_network/Data types/DATA_LOG/UNI_CIRCULAR_BUFFER_DATA.TcDUT
TYPE UNI_CIRCULAR_BUFFER_DATA :
STRUCT
	D_MODE : INT;
	D_HEAD : WORD;
	D_STRING : STRING(STRING_LENGTH);
	D_REAL : REAL;
	D_DWORD : DWORD;
	BUF_SIZE : UINT;
	BUF_COUNT : UINT;
	BUF_USED : USINT;
	BUF : NW_BUF_LONG;
	_GetStart : UINT;
	_GetEnd : UINT;
	_Last : UINT;
	_First : UINT;
END_STRUCT
END_TYPE

// ---- oscat_network/Data types/DATA_LOG/us_LOG_VIEWPORT.TcDUT
TYPE us_LOG_VIEWPORT :
STRUCT
	LINE_ARRAY : ARRAY [1..40] OF INT;
	COUNT : INT; (* Anzahl der sichtbaren Nachtrichten *)
	UPDATE_COUNT : UINT; (* Updatezähler *)
	MOVE_TO_X : INT; (* Steuerung der Nachrichtenanzeige *)
	UPDATE : BOOL; (* Daten wurden geändert -> neuzeichnen *)
END_STRUCT
END_TYPE

// ---- oscat_network/Data types/FILE_SERVER/FILE_PATH_DATA.TcDUT
TYPE FILE_PATH_DATA :
STRUCT
	DRIVE : STRING(3);
	DIRECTORY : STRING(STRING_LENGTH);
	FILENAME : STRING;
END_STRUCT
END_TYPE

// ---- oscat_network/Data types/FILE_SERVER/FILE_SERVER_DATA.TcDUT
TYPE FILE_SERVER_DATA :
STRUCT
	FILE_OPEN : BOOL;
	FILENAME : STRING;
	MODE : BYTE;
	OFFSET : UDINT;
	FILE_SIZE : UDINT;
	AUTO_CLOSE : TIME;
	ERROR : BYTE;
END_STRUCT
END_TYPE

// ---- oscat_network/Data types/NETWORK/IP2GEO_DATA.TcDUT
TYPE IP2GEO_DATA :
STRUCT
	STATE : BOOL;
	IP4 : DWORD;
	COUNTRY_CODE : STRING(2);
	COUNTRY_NAME : STRING(20);
	REGION_CODE : STRING(2);
	REGION_NAME : STRING(20);
	CITY : STRING(20);
	GEO_LATITUDE : REAL;
	GEO_LONGITUDE : REAL;
	TIME_ZONE_NAME : STRING(20);
	GMT_OFFSET : INT;
	IS_DST : BOOL;
END_STRUCT
END_TYPE

// ---- oscat_network/Data types/NETWORK/IP_C.TcDUT
TYPE IP_C :
STRUCT
	C_MODE : BYTE;						(*W Mode: TCP/UCP AKTIV/PASSIV                               *)
	C_PORT : WORD;						(*W Portnummer                                               *)
	C_IP : DWORD;						(*W IP-Adresse gepackt wwxxyyzz = www.xxx.yyy.zzz            *)
	C_STATE : BYTE;						(*R Verbindungsstatus ON/OFF + Flanke ON/OFF                 *)
	C_ENABLE : BOOL;					(*W Freigabe für Connect                                     *)
	R_OBSERVE : BOOL;					(*W Empfang ueberwachen                                      *)
	TIME_RESET : BOOL;					(*W Alle Timer ruecksetzen                                   *)
	ERROR : DWORD;					(*R vvwwxxyy (vv = CON_ERROR, ww = SEN_ERROR, xx = REC_ERROR *)
	FIFO : IP_FIFO_DATA;					(*I IP FIFO Struktur                                         *)
	MAILBOX : ARRAY [1..16] OF BYTE;	(*I Mailbox: Datenbereich für Bausteindatenaustausch         *)
END_STRUCT
END_TYPE

// ---- oscat_network/Data types/NETWORK/IP_FIFO_DATA.TcDUT
TYPE IP_FIFO_DATA :
STRUCT
	X : ARRAY [1..128] OF BYTE; 	(* IP_ID FIFO Speicher          *)
	Y : ARRAY [1..128] OF BYTE; 	(* IP_ID Zähler                 *)
	ID : BYTE;					(* höchste vergabene id         *)
	MAX_ID : BYTE;				(* maximal Anmeldungen pro ID   *)
	INIT : BOOL;					(* Initialisierung durchgeführt *)
	EMPTY : BOOL;				(* FIFO leer                    *)
	FULL : BOOL;					(* FIFO voll                    *)
	TOP : INT;					(* maximale anzahl in FIFO      *)
	NW : INT;					(* Schreibzeiger                *)
	NR : INT;						(* Lesezeiger                   *)
END_STRUCT
END_TYPE

// ---- oscat_network/Data types/NETWORK/NETWORK_BUFFER.TcDUT
TYPE NETWORK_BUFFER :
STRUCT
	SIZE : UINT;
	BUFFER : NW_BUF_LONG;
END_STRUCT
END_TYPE

// ---- oscat_network/Data types/NETWORK/NETWORK_BUFFER_SHORT.TcDUT
TYPE NETWORK_BUFFER_SHORT :
STRUCT
	SIZE : UINT;
	BUFFER : NW_BUF_SHORT;
END_STRUCT
END_TYPE

// ---- oscat_network/Data types/NETWORK/NW_BUF_LONG.TcDUT
TYPE
	NW_BUF_LONG  : ARRAY[0..NETWORK_BUFFER_LONG_SIZE] OF BYTE;
END_TYPE

// ---- oscat_network/Data types/NETWORK/NW_BUF_SHORT.TcDUT
TYPE
	NW_BUF_SHORT : ARRAY[0..NETWORK_BUFFER_SHORT_SIZE] OF BYTE;
END_TYPE

// ---- oscat_network/Data types/NETWORK/URL.TcDUT
TYPE URL :
STRUCT
	PROTOCOL : STRING(10);
	USER : STRING(32);
	PASSWORD : STRING(32);
	DOMAIN : STRING(80);
	PORT : WORD;
	PATH : STRING(80);
	QUERY : STRING(STRING_LENGTH);
	ANCHOR : STRING(40);
	HEADER : STRING(160);
END_STRUCT
END_TYPE

// ---- oscat_network/Data types/NETWORK/VMAP_DATA.TcDUT
TYPE VMAP_DATA :
STRUCT
	FC : DWORD;
	V_ADR : INT;
	V_SIZE : INT;
	P_ADR : INT;
	TIME_OUT : TIME;
END_STRUCT
END_TYPE

// ---- oscat_network/Data types/NETWORK/XML_CONTROL.TcDUT
TYPE XML_CONTROL :
STRUCT
	COMMAND : WORD;
	WATCHDOG : TIME;
	START_POS : UINT;
	STOP_POS : UINT;
	COUNT : UINT;
	TYP : INT;
	LEVEL : UINT;
	PATH : STRING(STRING_LENGTH);
	ELEMENT : STRING(STRING_LENGTH);
	ATTRIBUTE : STRING(STRING_LENGTH);
	VALUE : STRING(STRING_LENGTH);
	BLOCK1_START : UINT;
	BLOCK1_STOP : UINT;
	BLOCK2_START : UINT;
	BLOCK2_STOP : UINT;
END_STRUCT
END_TYPE

// ---- oscat_network/Data types/NET_VAR/NET_VAR_DATA.TcDUT
TYPE NET_VAR_DATA :
STRUCT
	CYCLE : UDINT;
	STATE : BYTE;
	INDEX : INT;
	ID_MAX : USINT;
	ERROR_ID : BYTE;
	BUF_SIZE : UINT;
	S_BUF : NETWORK_BUFFER;
	R_BUF : NETWORK_BUFFER;
END_STRUCT
END_TYPE

// ---- oscat_network/Data types/TELNET_VISION/us_TN_INPUT_CONTROL.TcDUT
TYPE us_TN_INPUT_CONTROL :
STRUCT
	bo_Enable: BOOL; (* Bearbeitung freigeben/sperren *)
	bo_Update_all: BOOL; (* All Elemente neu zeichnen *)
	bo_Reset_Fokus: BOOL; (* Fokus auf 1. Element setzen *)
	in_Focus_at: INT; (* Controlelement mit aktivem Fokus *)
	in_Count: INT; (* Anzahl der benutzen Control-Elemente *)
	in_ToolTip_X: INT; (* Tooltip Text X-Offset *)
	in_ToolTip_Y: INT; (* Tooltip Text Y-Offset *)
	by_ToolTip_Attr: BYTE; (* Tooltip Text Attribute *)
	in_ToolTip_Size: INT; (* Tooltip Text länge *)
	usa_TN_INPUT_CONTROL_DATA: ARRAY [1..20] OF us_TN_INPUT_CONTROL_DATA;
END_STRUCT
END_TYPE

// ---- oscat_network/Data types/TELNET_VISION/us_TN_INPUT_CONTROL_DATA.TcDUT
TYPE us_TN_INPUT_CONTROL_DATA :
STRUCT
 	by_Input_Exten_Code: BYTE;
	by_Input_ASCII_Code: BYTE;
	bo_Input_ASCII_IsNum: BOOL;
	in_Title_X_Offset: INT; (* Title Text X-Offset *)
	in_Title_Y_Offset: INT; (* Title Text Y-Offset *)
	by_Title_Attr: BYTE; (* Title Text Attribute *)
	st_Title_String: STRING; (* Title Text String *)
	in_Cursor_X: INT; (* aktuelle Cursor X-Position *)
	in_Cursor_Y: INT; (* aktuelle Cursor Y-Position *)
	in_Type: INT; (* Type des Elements *)
	in_X: INT; (* Element X-Position *)
	in_Y: INT; (* Element Y-Position *)
	in_Cursor_Pos: INT; (* aktuelle Cursorposition *)
	by_Attr_mF: BYTE; (* Text Attribute mit Fokus *)
	by_Attr_oF: BYTE; (* Text Attribute ohne Fokus *)
	in_selected: INT; (* Text Item wurde ausgewählt *)
	st_Input_Mask: STRING; (* Text Eingabemaske *)
	st_Input_Data: STRING(STRING_LENGTH); (* Text aktuelle Eingabedaten *)
	st_Input_String: STRING; (* Text Kopie nach Return-Taste *)
	st_Input_ToolTip: STRING; (* Text ToolTip (Eingabeinformation) *)
	in_Input_Option: INT; (* Text Ausgabe-Optionen *)
	bo_Input_Entered: BOOL; (* RETURN-Taste wurde betätigt *)
	bo_Input_Hidden: BOOL; (* Text versteckete Eingabe mit '*' *)
	bo_Input_Only_Num: BOOL; (* Text nur Nummerneingabe zulassen *)
	bo_Focus: BOOL; (* Element besitzt den Fokus *)
	bo_Update_Input: BOOL; (* Element wegen Benutzereingabe neuzeichnen *)
	bo_Update_All: BOOL; (* Element komplett neuzeichnen *)

END_STRUCT
END_TYPE

// ---- oscat_network/Data types/TELNET_VISION/us_TN_MENU.TcDUT
TYPE us_TN_MENU :
STRUCT
	st_Menu_Text: STRING(STRING_LENGTH); (* X Menue Texte *)
	in_Menu_E_Count: INT; (* Menue Elemente Anzahl *)
	in_Y: INT; (* Menue Zeilennummer  Y-Position *)
	in_X: INT; (* Menue Spaltennummer X-Position *)
	by_Attr_mF: BYTE; (* Text Attribute mit Fokus *)
	by_Attr_oF: BYTE; (* Text Attribute ohne Fokus *)
	in_X_SM_new: INT; (* neue Sub-Menu X-Position *)
	in_Y_SM_new: INT; (* neue Sub-Menu Y-Position *)
	in_X_SM_old: INT; (* alte Sub-Menu X-Position *)
	in_Y_SM_old: INT; (* alte Sub-Menu Y-Position *)
	in_Cur_Menu_Item: INT; (* aktuelles Haupt-Menue *)
	in_Cur_Sub_Item: INT; (* aktuelles Sub-Menue *)
	in_State: INT; (*   Menu status   *)
	in_Menu_Selected: INT; (* X Menu-Item mit Enter angewwählt *)
	bo_Create: BOOL; (* X Menu erzeugen *)
	bo_Destroy: BOOL; (* X Menu entfernen *)
	bo_Update: BOOL; (* X Menu updaten *)
END_STRUCT
END_TYPE

// ---- oscat_network/Data types/TELNET_VISION/us_TN_MENU_POPUP.TcDUT
TYPE us_TN_MENU_POPUP :
STRUCT
	st_Menu_Text: STRING(STRING_LENGTH); (* X Menue Texte *)
	in_Menu_E_Count: INT; (* Menue Elemente Anzahl *)
	in_X: INT; (* X Menue X-Position *)
	in_Y: INT; (* X Menue Y-Position *)
	in_Cols: INT; (* Menue Spaltenanzahl *)
	in_Rows: INT; (* Menue Zeilenanzahl *)
	in_Cur_Item: INT; (* X aktuelles Sub-Menue *)
	by_Attr_mF: BYTE; (* X Text Attribute mit Fokus	*)
	by_Attr_oF: BYTE; (* X Text Attribute ohne Fokus *)
	by_Input_Exten_Code: BYTE; (* X Tastencode: Sondertasten *)
	bo_Create: BOOL; (* X Popup-Menu erzeugen *)
	bo_Destroy: BOOL; (* X Popup-Menu entfernen *)
	bo_Update: BOOL; (* X Popup-Menu updaten *)
	bo_Activ: BOOL; (*   Popup-Menu ist aktiv *)
END_STRUCT
END_TYPE

// ---- oscat_network/Data types/TELNET_VISION/us_TN_SCREEN.TcDUT
TYPE us_TN_SCREEN :
STRUCT
	bya_CHAR: ARRAY [0..1919] OF BYTE;
	bya_COLOR: ARRAY [0..1919] OF BYTE;
	bya_BACKUP: ARRAY [0..1919] OF BYTE;
	bya_Line_Update: ARRAY [0..23] OF BOOL;
	by_Input_Exten_Code: BYTE;
	by_Input_ASCII_Code: BYTE;
	bo_Input_ASCII_IsNum: BOOL;
	in_Page_Number: INT; (* aktive Seiten-Nr. *)
	in_Cursor_X: INT; (* Cursor X-Position *)
	in_Cursor_Y: INT; (* Cursor Y-Position *)
	in_EOS_Offset: INT; (* End of String Offset *)
	by_Clear_Screen_Attr: BYTE; (* Clear-Screen Attr *)
	bo_Clear_Screen: BOOL; (* Clear-Screen auslösen *)
	bo_Modal_Dialog: BOOL; (* Modaler Dialog ist aktiv *)
	bo_Menue_Bar_Dialog: BOOL; (* Menue Dialog ist aktiv *)
END_STRUCT
END_TYPE

// ---- oscat_network/Data types/WEATHER/WORLD_WEATHER_CUR.TcDUT
TYPE WORLD_WEATHER_CUR :
STRUCT
	OBSERVATION_TIME : STRING(8);
	TEMP_C : INT;
	WEATHER_CODE : INT;
	WEATHER_DESC : STRING(60);
	WEATHER_ICON : INT;
	WIND_SPEED_MILES : INT;
	WIND_SPEED_KMPH : INT;
	WIND_DIR_DEGREE : INT;
	WIND_DIR16POINT : STRING(3);
	PRECIPMM : REAL;
	HUMIDITY : INT;
	VISIBILITY : INT;
	PRESSURE : INT;
	CLOUDOVER : INT;
END_STRUCT
END_TYPE

// ---- oscat_network/Data types/WEATHER/WORLD_WEATHER_DATA.TcDUT
TYPE WORLD_WEATHER_DATA :
STRUCT
	CUR : WORLD_WEATHER_CUR;
	DAY : ARRAY [0..4] OF WORLD_WEATHER_DAY;
END_STRUCT
END_TYPE

// ---- oscat_network/Data types/WEATHER/WORLD_WEATHER_DAY.TcDUT
TYPE WORLD_WEATHER_DAY :
STRUCT
	DATE_OF_DAY : STRING(10);
	TEMP_MAX_C : INT;
	TEMP_MAX_F : INT;
	TEMP_MIN_C : INT;
	TEMP_MIN_F : INT;
	WIND_SPEED_MILES : INT;
	WIND_SPEED_KMPH : INT;
	WIND_DIR_DEGREE : INT;
	WIND_DIR16POINT : STRING(3);
	WEATHER_CODE : INT;
	WEATHER_DESC : STRING(60);
	WEATHER_ICON : INT;
	PRECIPMM : REAL;
END_STRUCT
END_TYPE

// ---- oscat_network/Data types/WEATHER/YAHOO_WEATHER_DATA.TcDUT
TYPE YAHOO_WEATHER_DATA :
STRUCT
	TIMETOLIVE : INT;							(* TIME TO LIVE: HOW LONG IN MINUTES THIS FEED SHOULD BE CACHED         *)
	LOCATION_CITY : STRING(40);   				(* THE LOCATION OF THIS FORECAST: CITY: CITY NAME  *)
	LOCATION_REGION : STRING(20);  				(* THE LOCATION OF THIS FORECAST: REGION: STATE, TERRITORY, OR REGION, IF GIVEN *)
	LOCATION_COUNTRY : STRING(20);			(* THE LOCATION OF THIS FORECAST: COUNTRY: TWO-CHARACTER COUNTRY CODE *)
	UNIT_TEMPERATURE : STRING(1);				(* TEMPERATURE: DEGREE UNITS, F FOR FAHRENHEIT OR C FOR CELSIUS *)
	UNIT_DISTANCE : STRING(2);					(* DISTANCE: UNITS FOR DISTANCE, MI FOR MILES OR KM FOR KILOMETERS *)
	UNIT_PRESSURE : STRING(2);					(* PRESSURE: UNITS OF BAROMETRIC PRESSURE, IN FOR POUNDS PER SQUARE INCH OR MB FOR MILLIBARS *)
	UNIT_SPEED : STRING(4);						(* SPEED: UNITS OF SPEED, MPH FOR MILES PER HOUR OR KPH FOR KILOMETERS PER HOUR *)
	WIND_CHILL : INT;							(* FORECAST INFORMATION ABOUT WIND CHILL IN DEGREES *)
	WIND_DIRECTION : INT;						(* FORECAST INFORMATION ABOUT WIND DIRECTION, IN DEGREES *)
	WIND_SPEED : REAL;							(* FORECAST INFORMATION ABOUT WIND SPEED, IN THE UNITS (MPH OR KPH)*)
	ATMOSPHERE_HUMIDITY : INT;				(* FORECAST INFORMATION ABOUT CURRENT ATMOSPHERIC HUMIDITY: HUMIDITY, IN PERCENT  *)
	ATMOSPHERE_PRESSURE : INT;				(* FORECAST INFORMATION ABOUT CURRENT ATMOSPHERIC PRESSURE: BAROMETRIC PRESSURE, IN THE UNITS (IN OR MB) *)
	ATMOSPHERE_VISIBILITY : REAL;				(* FORECAST INFORMATION ABOUT CURRENT ATMOSPHERIC VISIBILITY, IN THE UNITS (MI OR KM) *)
	ATMOSPHERE_RISING : INT;					(* FORECAST INFORMATION ABOUT RISING: STATE OF THE BAROMETRIC PRESSURE: STEADY (0), RISING (1), OR FALLING (2). (INTEGER: 0, 1, 2) *)
	ASTRONOMY_SUNRISE : STRING(10);			(* SUNRISE: TODAY'S SUNRISE TIME. THE TIME IS A STRING IN A LOCAL TIME FORMAT OF "H:MM AM/PM" *)
	ASTRONOMY_SUNSET : STRING(10);			(* SUNSET: TODAY'S SUNSET TIME. THE TIME IS A STRING IN A LOCAL TIME FORMAT OF "H:MM AM/PM", *)
	GEO_LATITUDE : REAL;						(* THE LATITUDE OF THE LOCATION *)
	GEO_LONGITUDE : REAL;						(* THE LONGITUDE OF THE LOCATION *)
	CUR_CONDITIONS_TEMP : INT;				(* THE CURRENT WEATHER CONDITIONS: TEMP: THE CURRENT TEMPERATURE, IN THE UNITS (F OR C) *)
	CUR_CONDITIONS_TEXT : STRING(40);			(* THE CURRENT WEATHER CONDITIONS: TEXT: A TEXTUAL DESCRIPTION OF CONDITIONS *)
	CUR_CONDITIONS_CODE : INT;				(* THE CURRENT WEATHER CONDITIONS: CODE: THE CONDITION CODE FOR THIS FORECAST *)
	CUR_CONDITIONS_ICON : INT;					(* THE CURRENT WEATHER CONDITIONS: ICON: THE CONDITION ICON FOR THIS FORECAST *)
	FORCAST_TODAY_LOW_TEMP : INT;			(* THE FORCAST TODAY WEATHER CONDITIONS: THE FORECASTED LOW TEMPERATURE FOR THIS DAY IN THE UNITS (F OR C) *)
	FORCAST_TODAY_HIGH_TEMP : INT;			(* THE FORCAST TODAY WEATHER CONDITIONS: THE FORECASTED HIGH TEMPERATURE FOR THIS DAY IN THE UNITS (F OR C) *)
	FORCAST_TODAY_TEXT : STRING(40);			(* THE FORCAST TODAY WEATHER CONDITIONS: TEXT: A TEXTUAL DESCRIPTION OF CONDITIONS *)
	FORCAST_TODAY_CODE : INT;				(* THE CURRENT WEATHER CONDITIONS: CODE: THE CONDITION CODE FOR THIS FORECAST *)
	FORCAST_TODAY_ICON : INT;					(* THE CURRENT WEATHER CONDITIONS: ICON: THE CONDITION ICON FOR THIS FORECAST *)
	FORCAST_TOMORROW_LOW_TEMP : INT; 		(* THE FORCAST TOMORROW WEATHER CONDITIONS: THE FORECASTED LOW TEMPERATURE FOR THIS DAY IN THE UNITS (F OR C) *)
	FORCAST_TOMORROW_HIGH_TEMP : INT;		(* THE FORCAST TOMORROW WEATHER CONDITIONS: THE FORECASTED HIGH TEMPERATURE FOR THIS DAY IN THE UNITS (F OR C) *)
	FORCAST_TOMORROW_TEXT : STRING(40);	(* THE FORCAST TOMORROW WEATHER CONDITIONS: TEXT: A TEXTUAL DESCRIPTION OF CONDITIONS *)
	FORCAST_TOMORROW_CODE : INT;			(* THE CURRENT WEATHER CONDITIONS: CODE: THE CONDITION CODE FOR THIS FORECAST *)
	FORCAST_TOMORROW_ICON : INT;			(* THE CURRENT WEATHER CONDITIONS: ICON: THE CONDITION ICON FOR THIS FORECAST *)

END_STRUCT
END_TYPE

// ---- oscat_basic/Global Variables/Constants_2.TcGVL
{attribute 'Tc2GvlVarNames'}
VAR_GLOBAL CONSTANT
	STRING_LENGTH : INT := 250;
	LIST_LENGTH : INT := 250;
END_VAR




(* revisionhistory
hm 3. mar. 2007
	extended accuracy of pi2
	renamed T0 to Tk for better compatibility with other libraries
	renamed C t0 c0 for better compatibility

hm	2. may. 2007
	added RU universal gas constant

hm	1. oct. 2007
	added setup parameter STEP7

hm 31. oct. 2007
	added PN

hm	6. mar. 2008
	added setup Parameter EXTENDED_ASCII

hm	28. Mar. 2008
	added setup parameter STRING_LENGTH

hm	7. apr. 2008
	Deleted unused setup parameter Step7

hm	19. apr. 2008
	added setup parameter NETWORK_BUFFER_SIZE

hm	27. apr. 2008
	added PI05 and PI025

hm	18. may. 2008
	added charname lists
	renamed E to E1

hm	30. jun. 2008
	reduced size of string constants to 253 to avoid problems with target aixia DCUF

hm	21. sep. 2008
	added section language setup
	added section location setup

hm	20. oct. 2008
	changed to structured constants

hm	16. nov. 2008
	moved structured constants to global vars for compatibility reasons

hm	13. nov. 2009
	added network_buffer_short_size
	renamed network_buffer_long_size
	changed string length to 250

hm	20. jan. 2011
	removed network buffers
	added list_length
*)

// ---- oscat_building/Global Variables/Constants.TcGVL
{attribute 'Tc2GvlVarNames'}
VAR_GLOBAL CONSTANT
END_VAR

// ---- oscat_building/Global Variables/Setup_Data.TcGVL
{attribute 'Tc2GvlVarNames'}
VAR_GLOBAL RETAIN

END_VAR

// ---- oscat_network/Global Variables/Constants_1.TcGVL
{attribute 'Tc2GvlVarNames'}
VAR_GLOBAL CONSTANT
	NETWORK_BUFFER_LONG_SIZE : UINT := 4095;
	NETWORK_BUFFER_SHORT_SIZE : UINT := 1407;
	LOG_MAX : INT := 40;
	LOG_SIZE : INT := 80;
	ELEMENT_LENGTH : INT := 250;
END_VAR

// ---- oscat_network/Global Variables/Globale_Variablen_1.TcGVL
{attribute 'Tc2GvlVarNames'}
VAR_GLOBAL
	TCP_SERVER_RESET : BYTE; (* nur für TwinCAT notwendig ! *)
	LOG_CL : LOG_CONTROL;
END_VAR

// ---- oscat_basic/POUs/String/CHARNAME.TcPOU
FUNCTION CHARNAME : STRING(10)
VAR_INPUT
	C : BYTE;
END_VAR
VAR
	pos: INT;
	i : INT;
END_VAR

(*
version 1.4		17. dec. 2008
programmer 		hugo
tested by		oscat

CHARNAME converts a Character code into its HTML character name
ä is convterted to 'äuml'
€ is converted to 'euro'
the character itself is returned if no name is available for the character

*)

IF C <> 0 THEN
	(* construct search string from code followed by $ sign, also clear charname string*)
	CHARNAME := CHR_TO_STRING(C);
	CHARNAME := CONCAT(CHARNAME,'&');
	CHARNAME := CONCAT(';', CHARNAME);
	WHILE pos = 0 AND (i < 4) DO
		i := i + 1;
		pos := FIND(setup.CHARNAMES[i], CHARNAME);
	END_WHILE;
	IF pos > 0 THEN
		CHARNAME := MID(setup.CHARNAMES[i], 10, pos + 3);
		(* search for end of name and truncate *)
		pos := FIND(CHARNAME, ';');
		CHARNAME := LEFT(CHARNAME,pos - 1);
	ELSE
		CHARNAME := CHR_TO_STRING(C);
	END_IF;
ELSE
	CHARNAME := '';
END_IF;




(* revision history
hm	13. may. 2008	rev 1.0
	original version

hm	16. jun. 2008	rev 1.1
	changed nested call of concat for better compatibility

hm	19. oct. 2008	rev 1.2
	changes setup constants

hm	24. oct. 2008	rev 1.3
	new code for high performance

hm	17. dec. 2008	rev 1.4
	changed function chr to chr_to_string
*)

END_FUNCTION

// ---- oscat_basic/POUs/Buffer Management/BUFFER_SEARCH.TcPOU
FUNCTION BUFFER_SEARCH : INT
VAR_INPUT
	PT : POINTER TO ARRAY[0..32767] OF BYTE;
	SIZE : INT;
	STR : STRING(STRING_LENGTH);
	POS : INT;
	IGN : BOOL;
END_VAR
VAR
	ps : POINTER TO ARRAY[0..STRING_LENGTH] OF BYTE;
	chx : BYTE;
	i: INT;
	end: INT;
	k: INT;
	lx: INT;
END_VAR


(*
version 1.4	25. jan 2011
programmer 	hugo
tested by	oscat

this function will search for a string STR in an array of byte starting at position pos.
the function needs to be called: buffer_search(adr("array"),sizeof("array"), STR, POS, IGN);
because this function works with pointers its very time efficient and it needs no extra memory.
The function returns the position of the first character of the string in the array if found.
a -1 is returned if the string is not found in the array.
when IGN = TRUE, STR must be in capital letters and the search is case insensitv.

*)

ps := ADR(STR);
lx := LEN(STR);
end := MIN(SIZE - lx, SIZE - 1);
lx := lx - 1;
FOR i := pos TO end DO
	FOR k := 0 TO lx DO
		IF IGN THEN chx := TO_UPPER(pt^[i+k]); ELSE chx := pt^[i+k]; END_IF;
		IF ps^[k] <> chx THEN EXIT; END_IF;
	END_FOR;
	IF k > lx THEN
		BUFFER_SEARCH := i;
		RETURN;
	END_IF;
END_FOR;
BUFFER_SEARCH := -1;


(* revision History

hm 5. mar. 2008	rev 1.0
	original version

hm	16. mar. 2008	rev 1.1
	chaged type of input size to uint

hm	13. may. 2008	rev 1.2
	changed type of pointer to array[1..32767]
	changed size of string to STRING_LENGTH

hm	12. nov. 2009	rev 1.3
	limit end to array size

hm	25. jan. 2011	rev 1.4
	ign = True will now ignore case
	return -1 if nothing found
*)

END_FUNCTION

// ---- oscat_basic/POUs/Buffer Management/BUFFER_TO_STRING.TcPOU
FUNCTION BUFFER_TO_STRING : STRING(STRING_LENGTH)
VAR_INPUT
	PT : POINTER TO ARRAY[0..32767] OF BYTE;
	SIZE : UINT;
	START : UINT;
	STOP : UINT;
END_VAR
VAR
	ps : POINTER TO BYTE;
	i : UINT;
	stp: UINT;
	sta: UINT;
END_VAR


(*
version 1.5	12. nov. 2009
programmer 	hugo
tested by		oscat

this function will retrieve a string from an array of byte starting at position start and stop at position stop.
the function needs to be called:	buffer_TO_String(adr("array"),sizeof("array"), start, stop);
because this function works with pointers its very time efficient and it needs no extra memory.

*)

ps := ADR(BUFFER_TO_STRING);
IF size = 0 THEN RETURN; END_IF;
sta := MIN(start, size -1);
stp := MIN(stop, size -1);

(* check for maximum string_length *)
IF UINT_TO_INT(stp - sta + 1) >= STRING_LENGTH THEN
	stp := sta + INT_TO_UINT(STRING_LENGTH) - 1;
END_IF;

FOR i := sta TO stp DO
	ps^ := pt^[i];
	ps := ps + 1;
END_FOR;

(* terminate the string *)

ps^ := 0;



(* revision History
hm 	5. mar. 2008	rev 1.0
	original version

hm	16. mar. 2008	rev 1.1
	changed type of input size to uint

hm	13. may. 2008	rev 1.2
	changed type of pointer to array[0..32767]
	changed size of string to STRING_LENGTH

hm	12. jun. 2008	rev 1.3
	check for pointer overrun
	change input start and stop to uint
	added type conversions to avoid warnings under codesys 3.0

hm	23. mar. 2009	rev 1.4
	avoid writing to input stop

hm	12. nov. 2009 rev 1.5
	limit start and stop to size -1

*)

END_FUNCTION

// ---- oscat_basic/POUs/Buffer Management/_BUFFER_INSERT.TcPOU
FUNCTION _BUFFER_INSERT : INT
VAR_INPUT
	STR : STRING(STRING_LENGTH);
	POS : INT;
	PT : POINTER TO ARRAY[0..32767] OF BYTE;
	SIZE : UINT;
END_VAR
VAR
	end : INT;
	lx: INT;
	i: INT;
END_VAR


(*
version 1.5	2. jan. 2012
programmer 	hugo
tested by	oscat

this function will insert a string at a given position in a buffer.
the function needs to be called:	_buffer_init(adr("array"),sizeof("array"),init);
this function will manipulate a given array.
the function manipulates the original array, it returnes the next position after the input string when finished.
because this function works with pointers its very time efficient and it needs no extra memory.

*)

lx := LEN(str);
end := pos + lx;
(* first move the upper part of the buffer to make space for the string *)
FOR i := UINT_TO_INT(size) - 1 TO end BY -1 DO
	pt^[i] := pt^[i-lx];
END_FOR;
(* copy the string *)
_BUFFER_INSERT := _STRING_TO_BUFFER(str, pos, PT, size);


(* revision History
hm 	9. mar. 2008	rev 1.0
	original version

hm	16. mar. 2008	rev 1.1
	changed type of input size to uint

hm	13. may. 2008	rev 1.2
	changed type of pointer to array[1..32767]
	changed size of string to STRING_LENGTH

hm	23. mar. 2009	rev 1.3
	avoid writing to input pos

hm	12. nov. 2009	rev 1.4
	code optimized

hm 2. jan 2012	rev 1.5
	function now returns the next position after the input string

*)

END_FUNCTION

// ---- oscat_basic/POUs/Buffer Management/_BUFFER_UPPERCASE.TcPOU
FUNCTION _BUFFER_UPPERCASE : BOOL
VAR_INPUT
	PT : POINTER TO ARRAY[0..32000] OF BYTE;
	SIZE : INT;
END_VAR
VAR
	pos: INT;
END_VAR


(*
version 1.0	20. jan. 2011
programmer 	hugo
tested by	oscat

this function will convert an array of byte into uppercase
the function needs to be called:	_buffer_clear(adr("array"),sizeof("array"));
this function will manipulate a given array.
the function manipulates the original array, it rerturnes true when finished.
because this function works with pointers its very time efficient and it needs no extra memory.

*)

pos := 0;
WHILE pos < size DO
	PT^[pos] := TO_UPPER(pt^[pos]);
	pos := pos + 1;
END_WHILE;

_BUFFER_UPPERCASE := TRUE;

(* revision History
hm 	20. jan. 2011	rev 1.0
	original version

*)

END_FUNCTION

// ---- oscat_basic/POUs/Engineering/automation/DRIVER_1.TcPOU
FUNCTION_BLOCK DRIVER_1
VAR_INPUT CONSTANT
	Toggle_Mode : BOOL;
	Timeout : TIME;
END_VAR
VAR_INPUT
	SET : BOOL;
	IN : BOOL;
	RST : BOOL;
END_VAR
VAR_OUTPUT
	Q : BOOL;
END_VAR
VAR
	off : TON;
	edge: BOOL;
END_VAR

(*
version 1.0	2 jan 2008
programmer 	hugo
tested by		tobias

driver_1 is a multi purpose driver.
a rising edge on in sets the output high if toggle is flase. while toggle is true, a rising edge on in toggles the output Q.
if a timeout is specified the output q will be reset to false automatically after the timeout has elapsed.
a asynchronous reset and set will force the output high or low respectively.

*)

IF off.Q THEN Q := FALSE; END_IF;
IF rst THEN
	Q := FALSE;
ELSIF set THEN
	Q := TRUE;
ELSIF IN AND NOT edge THEN
	IF toggle_mode THEN q := NOT Q; ELSE q := TRUE; END_IF;
END_IF;
edge := in;
IF timeout > t#0s THEN off(in := Q, PT := Timeout); END_IF;


(* revision history
hm	2. jan 2008		rev 1.0
	original version

*)

END_FUNCTION_BLOCK

// ---- oscat_basic/POUs/Engineering/automation/FLOW_CONTROL.TcPOU
 FUNCTION_BLOCK FLOW_CONTROL
VAR_INPUT
	IN : BOOL;
	REQ : BOOL;
	ENQ : BOOL;
	RST : BOOL;
END_VAR
VAR_INPUT CONSTANT
	T_AUTO : TIME := T#1h;
	T_DELAY : TIME := T#23h;
END_VAR
VAR_OUTPUT
	Q : BOOL;
	STATUS : BYTE;
END_VAR
VAR
	timer : TP_1D;
END_VAR


(*
version 1.0	28. jun. 2008
programmer 	hugo
tested by	oscat

FLOW_CONTROL switches a valves depending on the input in.
flow control also limits the maximum ontime of the valve and controls pressure on the output side.

*)

STATUS := 100;
IF RST THEN
	Q := FALSE;
	timer(rst := TRUE);
	timer.RST := FALSE;
	STATUS := 103;
ELSIF ENQ THEN
	IF IN THEN
		status := 101;
	END_IF;
	IF REQ THEN
		(* timer will generate a timed pulse after TP goes high *)
		timer.PT1 := T_AUTO;
		timer.PTD := T_DELAY;
		timer.IN := TRUE;
		STATUS := 102;
	END_IF;
END_IF;


(* set output and run timer *)
timer();
timer.IN := FALSE;
Q := (IN AND ENQ) OR timer.Q;



(* revision history
hm 	28. jun. 2008 	rev 1.0
	original version

*)

END_FUNCTION_BLOCK

// ---- oscat_basic/POUs/Engineering/automation/INTERLOCK.TcPOU
FUNCTION_BLOCK INTERLOCK
VAR_INPUT
	I1, I2 : BOOL;
	TL : TIME;
END_VAR
VAR_OUTPUT
	Q1, Q2 : BOOL;
END_VAR
VAR
	T1, T2 : TOF;
END_VAR

(*
version 1.0	28 sep 2007
programmer 	hugo
tested by		tobias

INTERLOCK has two inputs I1 and I2 which drive the corresponding outputs Q1 and Q2.
the inputs signals lock each other out and therfore I1 can only drive Q1 when I2 is Low and vice versa.
The input TL specifies a dead time between two outputs can become active.
an output can only become active when the other output was not active for the time TL.

*)

(* the input signal have a run delay to lockout the other input *)
T1(IN := I1, PT := TL);
T2(IN := I2, PT := TL);

Q1 := I1 AND NOT t2.Q;
Q2 := I2 AND NOT t1.Q;


(* revision history

hm	28 sep 2007		rev 1.0
	original version

*)

END_FUNCTION_BLOCK

// ---- oscat_basic/POUs/Engineering/automation/INTERLOCK_4.TcPOU
FUNCTION_BLOCK INTERLOCK_4
VAR_INPUT CONSTANT
END_VAR
VAR_INPUT
	I0 : BOOL;
	I1 : BOOL;
	I2 : BOOL;
	I3 : BOOL;
	E : BOOL;
	MODE : INT;

END_VAR
VAR_OUTPUT
	OUT : BYTE;
	TP : BOOL;
END_VAR
VAR
	in: BYTE;
	last: BYTE;
	old: BYTE;
	lmode: INT;
END_VAR

(*
version 1.1	14. mar. 2009
programmer 	hugo
tested by		oscat

INTERLOCK_4 detects one of 4 switches and delivers the number of the switch pressed on the output out
a output tp is true for one cycle if the output has changed.
a setup variable MODE selects between 3 different modes:
MODE = 0, any input active will disable all other inputs
MODE = 1, the input with the highest number will be acepted
mode = 2, the input last pressed will disable all others 

*)

(* check if enable is active *)
IF E THEN
(* reset all vars when there is a mode change on thy fly *)
	IF mode <> lmode THEN
		out := 0;
		last := 0;
		old := 0;
		lmode := mode;
	END_IF;
	(* load inputs into in *)
	in.0 := I0;
	in.1 := I1;
	in.2 := I2;
	in.3 := I3;
	(* only execute when there is any change *)
	IF in <> last THEN
		(* only execute when inputs have chages state *)
		CASE mode OF
			0:	(* output directly display inputs as bits in byte out *)
				out := in;

			1:	(* the input with the highest number will be acepted *)
				IF in.3 THEN out := 8;
				ELSIF in.2 THEN out := 4;
				ELSIF in.1 THEN out := 2;
				ELSE out := in;
				END_IF;

			2:	(* input last pressed will be displayed only *)
				last := ((in XOR last) AND in);
				IF last.3 THEN out := 8;
				ELSIF last.2 THEN out := 4;
				ELSIF last.1 THEN out := 2;
				ELSE out := last;
				END_IF;

			3:	(* any input active will disable all other inputs *)
				IF (out AND in) = 0 THEN
					IF in.3 THEN out := 8;
					ELSIF in.2 THEN out := 4;
					ELSIF in.1 THEN out := 2;
					ELSE out := in;
					END_IF;
				END_IF;

		END_CASE;
		last := in;
	END_IF;
	tp := out <> old;
	old := out;
ELSE
	out := 0;
	last := 0;
	old := 0;
	lmode := 0;
	tp := FALSE;
END_IF;


(* revision history
hm	24. oct 2008	rev 1.0
	original version

hm	14. mar. 2009	rev 1.1
	replaced double assignments

*)

END_FUNCTION_BLOCK

// ---- oscat_basic/POUs/Engineering/automation/MANUAL.TcPOU
FUNCTION MANUAL : BOOL
VAR_INPUT
	IN : BOOL;
	ON : BOOL;
	OFF : BOOL;
END_VAR


(*
version 1.0	21. nov. 2008
programmer 	hugo
tested by	oscat

MANUAL is a manual override for digital signals.
when on and off = FALSE, the output follows IN.
ON = TRUE forces the output high, and OFF = TRUE forces the output low.


*)

MANUAL := NOT OFF AND (IN OR ON);



(* revision history
hm	21. nov 2008	rev 1.0
	original version


*)

END_FUNCTION

// ---- oscat_basic/POUs/Engineering/automation/MANUAL_1.TcPOU
FUNCTION_BLOCK MANUAL_1
VAR_INPUT
	IN : BOOL;
	MAN : BOOL;
	M_I : BOOL;
	SET : BOOL;
	RST : BOOL;
END_VAR
VAR_OUTPUT
	Q : BOOL;
	STATUS : BYTE;
END_VAR
VAR
	S_edge : BOOL;
	r_edge : BOOL;
	edge: BOOL;
END_VAR

(*
version 1.2	14. mar. 2009
programmer 	hugo
tested by		oscat

MANUAL_1 is a manual override for digital signals.
When MAN = FALSE, the output follows IN and when MAN = TRUE the Output follows M_I.


*)

IF NOT man THEN
	Q := IN;
	STATUS := 100;
	edge := FALSE;
ELSIF NOT s_edge AND set THEN
	Q := TRUE;
	edge := TRUE;
	status := 101;
ELSIF NOT r_edge AND rst THEN
	Q := FALSE;
	edge := TRUE;
	status := 102;
ELSIF NOT edge THEN
	Q := M_I;
	status := 103;
END_IF;

(* remember levels of manual signals *)
s_edge := SET;
r_edge := RST;



(* revision history
hm	17. jun 2008	rev 1.0
	original version

hm	17. oct 2008	rev 1.1
	deleted unnecessary variable m_edge

hm	14. mar. 2009	rev 1.2
	replaced double assignments

*)

END_FUNCTION_BLOCK

// ---- oscat_basic/POUs/Engineering/automation/PARSET2.TcPOU
FUNCTION_BLOCK PARSET2
VAR_INPUT
	X : REAL;
END_VAR
VAR_INPUT CONSTANT
	X01, X02, X03, X04 : REAL;
	X11, X12, X13, X14 : REAL;
	X21, X22, X23, X24 : REAL;
	X31, X32, X33, X34 : REAL;
	L1, L2, L3 : REAL;
	TC : TIME;
END_VAR
VAR_OUTPUT
	P1,P2,P3,P4 : REAL;
END_VAR
VAR
	Pset : parset;
	init: BOOL;
END_VAR

(*
version 1.0	3 nov 2007
programmer 	hugo
tested by	tobias

parset2 selects on of 4 parameter sets depending on the value of X. if TC is specified, the change of the outputs
is ramped by the time TC
*)

(* init sequence *)
IF NOT init THEN
	init := TRUE;
	pset(TC:=TC, X01:=X01, X02:=X02, X03:=X03, X04:=X04, X11:=X11, X12:=X12, X13:=X13, X14:=X14, X21:=X21, X22:=X22, X23:=X23, X24:=X24, X31:=X31, X32:=X32, X33:=X33, X34:=X34);
END_IF;
IF ABS(X) < L1 THEN
	pset(A0 := FALSE, A1 := FALSE);
ELSIF ABS(X) < L2 THEN
	pset(A0 := TRUE, A1 := FALSE);
ELSIF ABS(x) < L3 THEN
	pset(A0 := FALSE, A1 := TRUE);
ELSE
	pset(A0 := TRUE, A1 := TRUE);
END_IF;
P1 := pset.P1;
P2 := pset.P2;
P3 := pset.P3;
P4 := pset.P4;

(* revision history
hm		3.11.2007		rev 1.0
	original version

*)

END_FUNCTION_BLOCK

// ---- oscat_basic/POUs/Engineering/automation/SIGNAL_4.TcPOU
FUNCTION_BLOCK SIGNAL_4
VAR_INPUT
	IN1 : BOOL;
	IN2 : BOOL;
	IN3 : BOOL;
	IN4 : BOOL;
	TS : TIME;
END_VAR
VAR_INPUT CONSTANT
	S1 : BYTE := 2#1111_1111;
	S2 : BYTE := 2#1111_0000;
	S3 : BYTE := 2#1010_1010;
	S4 : BYTE := 2#1010_0000;
END_VAR
VAR_OUTPUT
	Q : BOOL;
END_VAR
VAR
	sig : SIGNAL;
END_VAR

(*
version 1.0	13 dec 2007
programmer 	hugo
tested by		tobias

this function generates one out of 4 signals specified by bit patterns S1 .. S4.
the selected pattern will be shifted with the step time TS.
In1 has higher priority then In2 which has higher priority then IN3 and in4 has the lowest priority.
ts defaults to 128 ms if not specified.
*)

(* an alarm is present read system time first *)
(* check if an alarm is present if yes set sig to the alarm pattern otherwise exit the routine *)
IF in1 THEN
	sig(in := TRUE, sig := s1, TS := TS);
ELSIF in2 THEN
	sig(in := TRUE, sig := s2, TS := TS);
ELSIF in3 THEN
	sig(in := TRUE, sig := s3, TS := TS);
ELSIF in4 THEN
	sig(in := TRUE, sig := s4, TS := TS);
ELSE
	sig(in := FALSE);
END_IF;

(* set the output *)
Q := sig.Q;


(* revision history
hm	13.12.2007		rev 1.0
	original version

*)

END_FUNCTION_BLOCK

// ---- oscat_basic/POUs/Engineering/Control/CONTROL_SET1.TcPOU
FUNCTION_BLOCK CONTROL_SET1
VAR_INPUT
	Kt : REAL;
	Tt : REAL;
	PI : BOOL;
	PID : BOOL;
END_VAR
VAR_INPUT CONSTANT
	P_K : REAL := 0.5;
	PI_K : REAL := 0.45;
	PI_TN : REAL := 0.83;
	PID_K : REAL := 0.6;
	PID_TN : REAL := 0.5;
	PID_TV : REAL := 0.125;
END_VAR
VAR_OUTPUT
	KP : REAL;
	TN : REAL;
	TV : REAL;
	KI : REAL;
	KD : REAL;
END_VAR


(*
version 1.1	11. mar. 2009
programmer 	hugo
tested by		tobias

takahashi calculates controller parameters for P, PI and PID controllers based on the ziegler nichols method.

*)

IF pi AND PID THEN
	KP := 0.0;
	TN := 0.0;
	TV := 0.0;
ELSIF PID THEN
	KP := PID_K * Kt;
	TN := PID_TN * Tt;
	TV := PID_TV * Tt;
ELSIF PI THEN
	KP := PI_K * Kt;
	TN := PI_TN * Tt;
ELSE
	KP := P_K * Kt;
END_IF;

(* KI and KD are calculated *)
IF tn > 0.0 THEN KI := KP / TN; ELSE KI := 0.0; END_IF;
KD := KP * TV;

(* revision history
hm	4. nov 2007	rev 1.0
	original version

hm	11. mar. 2009	rev 1.1
	real constants updated to new systax using dot																																																																																																																																																																																																																																																																																																																																																																																																																																																																																																																																																																																																																																																																																																																																																																																																																																																																																																																																																																																																																																																											

*)

END_FUNCTION_BLOCK

// ---- oscat_basic/POUs/Engineering/Control/CONTROL_SET2.TcPOU
FUNCTION_BLOCK CONTROL_SET2
VAR_INPUT
	KS : REAL;
	TU : REAL;
	TG : REAL;
	PI : BOOL;
	PID : BOOL;
END_VAR
VAR_INPUT CONSTANT
	P_K : REAL := 1.0;
	PI_K : REAL := 0.9;
	PI_TN : REAL := 3.33;
	PID_K : REAL := 1.2;
	PID_TN : REAL := 2.0;
	PID_TV : REAL := 0.5;
END_VAR
VAR_OUTPUT
	KP : REAL;
	TN : REAL;
	TV : REAL;
	KI : REAL;
	KD : REAL;
END_VAR
VAR
	TX : REAL;
END_VAR

(*
version 1.1	11. mar. 2009
programmer 	hugo
tested by		tobias

takahashi calculates controller parameters for P, PI and PID controllers based on the ziegler nichols method.

*)

IF TU > 0.0 AND KS > 0.0 THEN TX := TG / TU / KS; END_IF;
IF pi AND PID THEN
	KP := 0.0;
	TN := 0.0;
	TV := 0.0;
ELSIF PID THEN
	KP := PID_K * TX;
	TN := PID_TN * TU;
	TV := PID_TV * TU;
ELSIF PI THEN
	KP := PI_K * TX;
	TN := PI_TN * TU;
ELSE
	KP := P_K * TX;
END_IF;

(* KI and KD are calculated *)
IF TN > 0.0 THEN KI := KP / TN; ELSE KI := 0.0; END_IF;
KD := KP * TV;

(* revision history
hm	4. nov 2007	rev 1.0
	original version

hm	11. mar. 2009	rev 1.1
	real constants updated to new systax using dot																																																																																																																																																																																																																																																																																																																																																																																																																																																																																																																																																																																																																																																																																																																																																																																																																																																																																																																																																																																																																																																											

*)

END_FUNCTION_BLOCK

// ---- oscat_basic/POUs/Engineering/Control/CTRL_IN.TcPOU
FUNCTION CTRL_IN : REAL
VAR_INPUT
	SET_POINT, ACTUAL, NOISE : REAL;
END_VAR


(*
version 1.0	2. jun 2008
programmer 	hugo
tested by		tobias


*)

(* calculate the process error DIFF *)
CTRL_IN := DEAD_ZONE(SET_POINT - ACTUAL, NOISE);


(* revision history
hm 	2. jun. 2008 	rev 1.0
	original version

*)

END_FUNCTION

// ---- oscat_basic/POUs/Engineering/Control/CTRL_OUT.TcPOU
FUNCTION_BLOCK CTRL_OUT
VAR_INPUT
	CI, OFFSET, MAN_IN, LIM_L, LIM_H : REAL;
	MANUAL : BOOL;
END_VAR
VAR_OUTPUT
	Y : REAL;
	LIM : BOOL;
END_VAR


(*
version 1.1	5. nov 2008
programmer 	hugo
tested by	oscat


*)

Y := SEL(MANUAL, CI, MAN_IN) + OFFSET;

(* Limit the output *)
IF Y > LIM_L AND Y < LIM_H THEN
	LIM := FALSE;
ELSE
	Y := LIMIT(LIM_L, Y, LIM_H);
	LIM := TRUE;
END_IF;



(* revision history
hm 	2. jun. 2008 	rev 1.0
	original version

hm	5. nov. 2008	rev 1.1
	optimized code
*)

END_FUNCTION_BLOCK

// ---- oscat_basic/POUs/Engineering/Control/CTRL_PI.TcPOU
FUNCTION_BLOCK CTRL_PI
VAR_INPUT
	ACT, SET, SUP, OFS, M_I : REAL;
	MAN : BOOL;
	RST : BOOL;
	KP : REAL := 1.0;
	KI : REAL := 1.0;
	LL : REAL := -1000.0;
	LH : REAL := 1000.0;
END_VAR
VAR_OUTPUT
	Y : REAL;
	DIFF : REAL;
	LIM : BOOL;
END_VAR
VAR
	pi : FT_PIWL;
	co : CTRL_OUT;
END_VAR

(*
version 2.0	30. jun 2008
programmer 	hugo
tested by	oscat

FT_PI is a PI controller with manual functionality.
The PID controller works according to the fomula Y = e *(KP+ KI * INTEG(e) ) + offset, while e = set_point - actual.
a rst will reset all internal data, while a switch to manual will cause the controller to follow the function Y = manual_in + offset.
limit_h and Limit_l set the possible output range of Y.
the output flags lim will signal that the output limits are active and overflow will signal that the integrator has reached its limits.

since rev 1.1 the "trapezregel is used for more accuracy.
rev 1.2 added selective integratin which means the integrative component is only active within a small range of the target value 
this avoids the integrator to go to limits while an input setpoint change happened and is only causing overshoots.
the int_band is by default 100 which means the int is active all the time and if set to for example to 0.1 the integrator is only active
while the input is between 0.9 and 1.1 of the set_point value.

default values for KP = 1, TN = 1, TV = 1, LIMIT_L = -1000, LIMIT_H = +1000.
*)

DIFF := CTRL_IN(SET, ACT, SUP);
pi(in := DIFF, kp := KP, ki := KI, lim_l := LL, lim_h := LH, rst := RST);
co(ci := pi.Y, OFFSET := OFS, man_in := M_I, lim_l := LL, lim_h := LH, MANUAL := MAN);
Y := co.Y;
LIM := co.LIM;


(* revision history
hm 	31.10.2007 		rev 1.0
	original version

hm	3.11.2007		rev 1.1
	added noise input to filter noise
	added output diff
	set limit output false when output is within limits
	overfolw was not set correctly

hm	5. jan 2008		rev 1.2
	improved performance

hm	20. jun. 2008	rev 2.0
	rewritten using new modular approach

*)

END_FUNCTION_BLOCK

// ---- oscat_basic/POUs/Engineering/Control/CTRL_PID.TcPOU
FUNCTION_BLOCK CTRL_PID
VAR_INPUT
	ACT, SET, SUP, OFS, M_I : REAL;
	MAN : BOOL;
	RST : BOOL;
	REV : BOOL := FALSE;
	KP : REAL := 1.0;
	TN : REAL := 1.0;
	TV : REAL := 1.0;
	LL : REAL := -1000.0;
	LH : REAL := 1000.0;
END_VAR
VAR_OUTPUT
	Y : REAL;
	DIFF : REAL;
	LIM : BOOL;
END_VAR
VAR
	pid : FT_PIDWL;
	co : CTRL_OUT;
END_VAR



(*
version 2.0	30. jun. 2008
programmer 	hugo
tested by	oscat

FT_PI is a PI controller with manual functionality.
The PID controller works according to the fomula Y = e *(KP+ KI * INTEG(e) ) + offset, while e = set_point - actual.
a rst will reset all internal data, while a switch to manual will cause the controller to follow the function Y = manual_in + offset.
limit_h and Limit_l set the possible output range of Y.
the output flags lim will signal that the output limits are active.

*)

IF REV THEN
	DIFF := CTRL_IN(ACT, SET, SUP);
ELSE
	DIFF := CTRL_IN(SET, ACT, SUP);
END_IF
pid(in := DIFF, kp := KP, tn := TN, tv := TV, lim_l := LL, lim_h := LH, rst := RST);
co(ci := pid.Y, OFFSET := OFS, man_in := M_I, lim_l := LL, lim_h := LH, MANUAL := MAN);
Y := co.Y;
LIM := co.LIM;


(* revision history

hm 1.12.2006	 	rev 1.1
	changed algorithm to trapezregel for higher accuracy.

hm 3.1.2007		rev 1.2
	added integ_band to select when the integrator is active.

hm	3.3.2007		rev 1.3
	added default values to inputs KP, TN, TV, LIMIT_L und LIMIT_H.

hm 31.oct 2007	rev 1.4
	total rewrite of the module to avoid failures when one of the limits is 0

hm	3.11.2007	rev 1.5
	added noise input to filter noise
	added output diff
	set limit output false when output is within limits
	overfolw was not set correctly

hm	5. jan 2008	rev 1.6
	improved code for better performance
	
PhOstmann 09. nov 2020 rev 2.1
	added the possibility to reverse the control input difference
*)

END_FUNCTION_BLOCK

// ---- oscat_basic/POUs/Engineering/Control/FT_PIDWL.TcPOU
FUNCTION_BLOCK FT_PIDWL
VAR_INPUT
	IN : REAL;
	KP : REAL := 1.0;
	TN : REAL := 1.0;
	TV : REAL := 1.0;
	LIM_L : REAL := -1.0E38;
	LIM_H : REAL := 1.0E38;
	RST : BOOL;
END_VAR
VAR_OUTPUT
	Y : REAL;
	LIM : BOOL;
END_VAR
VAR
	piwl : FT_PIWL;
	diff : FT_DERIV;
END_VAR

(*
version 1.3	13. nov. 2009
programmer 	hugo
tested by		tobias

FT_PIDWL is a PID controller with dynamic wind_up reset.
The PID controller works according to the fomula Y = KP *(IN + KI * INTEG(e) + DERIV(e) ).
a rst will reset the integrator to 0
lim_h and Lim_l set the possible output range of the internal integrator.
the output flags lim will signal that the output limits are active.

default values for KP = 1, KI = 1, ILIM_L = -1E37, iLIM_H = +1E38.
*)

(* if rst then *)
IF rst THEN
	piwl(rst := TRUE);
	piwl.RST := FALSE;
ELSE
	(* run PIWL controller first *)
	(* we need to check if TN = 0 and do alternative calls *)
	IF TN = 0.0 THEN
		piwl(in := IN * KP, KP := 1.0, KI := 0.0, LIM_L := LIM_L, LIM_H := LIM_H);
	ELSE
		piwl(in := IN * KP, KP := 1.0, KI := 1.0 / TN, LIM_L := LIM_L, LIM_H := LIM_H);
	END_IF;

	(* run differentiator and add_to_output *)
	diff(IN := IN, K := KP * TV);
	Y := piwl.Y + diff.out;

	(* limit the output *)
	IF Y < LIM_L THEN
		LIM := TRUE;
		Y := LIM_L;
	ELSIF Y > LIM_H THEN
		LIM := TRUE;
		Y := LIM_H;
	ELSE
		LIM := FALSE;
	END_IF;
END_IF;



(* revision history
hm 13. jun. 2008 	rev 1.0
	original version

hm	25. jan 2008	rev 1.1
	multiply differential part with KP

hm	11. mar. 2009	rev 1.2
	real constants updated to new systax using dot

hm	13. nov. 2009	rev 1.3
	fixed code for negative KP

*)

END_FUNCTION_BLOCK

// ---- oscat_basic/POUs/Engineering/Control/DEAD_BAND_A.TcPOU
FUNCTION_BLOCK DEAD_BAND_A
VAR_INPUT
	X : REAL;
	T : TIME;
	KL : REAL := 1.0;
	LM : REAL;
END_VAR
VAR_OUTPUT
	Y : REAL;
	L : REAL;
END_VAR
VAR
	tp1 : FT_PT1;
	tp2 : FT_PT1;
END_VAR


(*
version 1.1	11. mar. 2009
programmer 	hugo
tested by		oscat

DEAD_BAND ist eine lineare Übertragungsfunktion mit Totzone. Die Funktion verschiebt den positiven Teil der Kurve um -L und den negativen Teil der Kurve um +L.
DEAD_BAND = X wenn Abs(X) > L wenn Abs(X) > L
DEAD_BAND = 0 wenn Abs(X) <= L
Die Breite der Totzone wird automatisch aus dem Signalrauschen errechnet.

*)

(* filter the input signal *)
tp1(in := X, T:= T);

(* filter the HF portion to generate a stable L *)
tp2(in := ABS(tp1.out - X), T := MULTIME(T, 4.0));

(* now we determine L which is half the width of the dead band *)
L := MIN(KL * tp2.out, LM);

IF X > L THEN
	Y := X - L;
ELSIF X < -L THEN
	Y := X + L;
ELSE
	Y := 0.0;
END_IF;


(* revision history
hm	14. jun. 2008	rev 1.0
	original version

hm	11. mar. 2009	rev 1.1
	real constants updated to new systax using dot

*)

END_FUNCTION_BLOCK

// ---- oscat_basic/POUs/Engineering/Control/FT_PT1.TcPOU
FUNCTION_BLOCK FT_PT1
VAR_INPUT
	in : REAL;
	T : TIME;
	K : REAL := 1.0;
END_VAR
VAR_OUTPUT
	out : REAL;
END_VAR
VAR
	last : DWORD;
	tx: DWORD;
	init: BOOL;
END_VAR

(*
version 1.11	18. jan. 2011
programmer 	hugo
tested by		oscat

FT_PT1 is an low pass filter with a programmable time T and faktor K.
 
*)

(* read system time *)
tx := T_PLC_US();

(* startup initialisation *)
IF NOT init OR T = t#0s THEN
	init := TRUE;
	out := K * in;
ELSE
	out := out + (in * K - out) * DWORD_TO_REAL(Tx - last) / TIME_TO_REAL(T) * 1.0E-3;
	IF ABS(out) < 1.0E-20 THEN out := 0.0; END_IF;
END_IF;
last := tx;


(*
hm 1.1.2007	rev 1.1
	corrected error while startup value was not correct
	for very small time values real output would run out of range.

hm 3.1.2007	rev 1.2
	corrected an error for falling edge failures.
	added output faktor K.

hm 27. 2. 2007	rev 1.3
	output will be input during init for definitive startup condition.

hm	15.9.2007	rev 1.4
	changed time() to T_PLC_US() for compatibilitxy resons
	increased internal accuracy to Microseconds instead of Milliseconds

hm	23. oct 2007	rev 1.5
	added out := in to the init statements

hm	30. nov 2007	rev 1.6
	changed out to be K * in during initialization

hm	5. jan 2008	rev 1.7
	improved code for better performance

hm	16. mar. 2008	rev 1.8
	added type conversion to avoid warning under codesys 3.0

hm	14. jun. 2008	rev 1.9
	improved code

hm	11. mar. 2009	rev 1.10
	real constants updated to new systax using dot

hm	18. jan. 2011	rev 1.11
	avoid underrun of out
*)

END_FUNCTION_BLOCK

// ---- oscat_basic/POUs/Engineering/measurements/T_PLC_US.TcPOU
FUNCTION T_PLC_US : DWORD
VAR CONSTANT
	debug : BOOL := 0;
	N : INT := 0;
	offset : DWORD := 0;
END_VAR
VAR
	tx : TIME;
END_VAR

(*
version 1.2	16 nov 2008
programmer 	hugo
tested by	tobias

T_PLC_US reads the internal PLC timer and return the time, it has the advantage to be able to set a debug mode 
and speed up the counter to test the plc timer overrun which occurs every 50 days respectively 25 days at siemens S7
this routine also allows to correct the behavior of s7 where the internal plc counter will not count all 32 bits.

*)

tx := TIME();
T_PLC_US := TIME_TO_DWORD(Tx)*1000;
(* hier muss die korrektur für step7 stattfinden
plctime muss den vollen wertebereich von time ausnutzen:
wenn bei step7 time -24tage bis plus 24 tage ist dann muss der timer auch beim überlauf auf -24tage springen 
und auf keinen fall auf 0 !!!!
für siemens muss ein weiterer fb im main eingebunden werden der sicherstellt das alle 32 bits durchgezählt werden.
es kann nur ein fb sein den er muss sich das oberste (32te) bit merken.
oder etwa spring s7 bei überlauf auf -24 tage????? dann wäre keine korrektur nötig.
*)
IF debug THEN
	T_PLC_US := (SHL(T_PLC_US,N) OR SHL(DWORD#1,N)-1) + OFFSET;
END_IF;

(* revision history
hm	14.9.2007	rev 1.0
	original version

hm	12. nov 2007	rev 1.1
	added temporaray variable tx because some compilers could not handle time() as an argument

hm	16. nov. 2008	rev 1.2
	initialized constants with 0 for compatibility reasons

*)

END_FUNCTION

// ---- oscat_basic/POUs/Time&Date/MULTIME.TcPOU
FUNCTION MULTIME : TIME
VAR_INPUT
	t : TIME;
	M : REAL;
END_VAR


(*
version 1.1	14 mar 2008
programmer 	hugo
tested by		tobias

multiplies a time by a real number and returns a time
*)

MULTIME := DWORD_TO_TIME(REAL_TO_DWORD(DWORD_TO_REAL(TIME_TO_DWORD(t))*M));

(* revision history
hm		2. oct 2006	rev 1.0
	original version

hm		14. mar 2008	rev 1.1
	rounded the result after the last digit

*)

END_FUNCTION

// ---- oscat_basic/POUs/Engineering/Control/VOLTAGE_CONTROL.TcPOU
FUNCTION_BLOCK VOLTAGE_CONTROL EXTENDS FB_CONTROL 
VAR
	fbOutput		: FB_OutLinear;
END_VAR

METHOD Control
IF fSet < 0 THEN
	fSet := 0;
END_IF

SUPER^.Control();
END_METHOD

PROPERTY Output : REFERENCE TO FB_OutLinear
GET
Output REF=THIS^.fbOutput;
END_GET
END_PROPERTY

METHOD Write
fbOutput.ValueOut := SUPER^.fY;
IF fSet <= 0 THEN
	fbOutput.ValueOut := 0;
END_IF
fbOutput.Write();
END_METHOD

END_FUNCTION_BLOCK

// ---- oscat_basic/POUs/Engineering/Control/FB_CONTROL.TcPOU
FUNCTION_BLOCK FB_CONTROL
VAR
	//Properties
	eControlMode		: CONTROL_MODE;
	stControlParameter	: CONTROL_PARAMETERS;
	
	fAct		:	REAL; 	// act value
	fSet		:	REAL; 	// set value
	fY			:	REAL; 	// control difference
	
	fbPID	:	FB_PID;
END_VAR

PROPERTY Act : REAL
GET
Act:=THIS^.fAct;
END_GET
SET
THIS^.fAct:=Act;
END_SET
END_PROPERTY

METHOD Control
VAR
	bResetController	: BOOL := FALSE;
END_VAR
IF fSet > 0 THEN
	bResetController := FALSE;
	// PID parameters are set in GVL 'ControlParameter_Props'
	fbPID(
		xSet := fSet,
		xAct := fAct,
		Kp := ControlParameter.Kp,
		Ti := ControlParameter.Ti,
		Td := ControlParameter.Td,
		LimLow := ControlParameter.LimLow,
		LimHigh := ControlParameter.LimHigh,
		bReverseActing := ControlParameter.bReverseActing,
		RST := bResetController,
		Y => fY
		);
ELSE
	IF NOT bResetController THEN
		bResetController := TRUE;
		fbPID(
		xSet := fSet,
		xAct := fAct,
		Kp := ControlParameter.Kp,
		Ti := ControlParameter.Ti,
		Td := ControlParameter.Td,
		LimLow := ControlParameter.LimLow,
		LimHigh := ControlParameter.LimHigh,
		bReverseActing := ControlParameter.bReverseActing,
		RST := bResetController,
		Y => fY
		);
	END_IF
	fY := 0;
END_IF
END_METHOD

PROPERTY ControlMode : CONTROL_MODE
GET
ControlMode := THIS^.eControlMode;
END_GET
SET
THIS^.eControlMode := ControlMode;
END_SET
END_PROPERTY

PROPERTY ControlParameter : REFERENCE TO CONTROL_PARAMETERS
GET
ControlParameter REF=THIS^.stControlParameter;
END_GET
SET
THIS^.stControlParameter := ControlParameter;
END_SET
END_PROPERTY

PROPERTY Set : REAL
GET
Set:=THIS^.fSet;
END_GET
SET
THIS^.fSet:=Set;
END_SET
END_PROPERTY

PROPERTY Y : Real
GET
Y :=THIS^.fY;
END_GET
END_PROPERTY

END_FUNCTION_BLOCK

// ---- oscat_basic/POUs/Engineering/Control/FB_PID.TcPOU
FUNCTION_BLOCK FB_PID
(* This PID controller implements an integrator anti-windup method (back-calculation). 
For this the difference between the unlimited control output the limited control output is added to the integrator input. 
This is done continously, allowing to track and correct the gain of the integrator.
*)
VAR_INPUT
	xSet:	REAL; 	// Set value
	xAct:	REAL;	// measured Value	

	Kp  :  	REAL;  	// proportional factor
	Ti  :  	REAL;  	// integral time
	Td  :	REAL; 	// derivative time
	Ni  :	REAL := 0.9; 	// time for anti-wiundup compensation
		
	LimLow	:	REAL; 	// lower limit of output
	LimHigh	: 	REAL; 	// upper limit of output
	StartY	:	REAL;	// Y to use as offset
	
	bReverseActing 	:	BOOL;	// True for reverse acting
	
	RST		:	BOOL; 	// True, if integrator should be resetted
	inStart	:	REAL := 0; 	// Value to which Integrator is resetted if RST is True
END_VAR
VAR_OUTPUT
	Y : REAL;		// controller output
	LIM : BOOL;		// True, if output reaches LimLow or LimHigh
END_VAR
VAR
	e			 :  REAL;		// control difference
	yOffset		 :  REAL	:= 0;		// constant offset used on Y	
	fbDerivative :  FT_DERIV; 	// function block for derivation
	fbIntegrate  :	FB_Integrate;	// function block for integration
	
	e_gaintrack	:  REAL;		// control difference for integrator
	Y_gaintrack	:  REAL := 0;	// tracking gain of y for Anti-windup
END_VAR

IF StartY <> yOffset THEN
	yOffset := StartY;
	fbIntegrate(RST:=TRUE, inStart:=inStart);
END_IF
IF RST THEN
	fbIntegrate(RST:=TRUE, inStart:=inStart);
END_IF

//determine direct or reverse acting
IF bReverseActing THEN
	e := xAct - xSet;
ELSE
	e := xSet - xAct;	
END_IF;

// correct control for integrator error based on previous integrations
e_gaintrack := e + Y_gaintrack/(Kp*Ni);

IF Ti>0 THEN
	//derivative and integral calculation
	fbDerivative(in:=e,run:=TRUE);
	fbIntegrate(run:= TRUE, in := e_gaintrack, RST:=RST);
	Y := Kp * (e + 1/Ti * fbIntegrate.out + Td * fbDerivative.out) + yOffset;
ELSE
	//derivative  calculation
	fbDerivative(in:=e,run:=TRUE);
	Y := Kp * (e + Td * fbDerivative.out) + yOffset;
END_IF

// check limits and track gain for adjusting next control error of integrator
IF Y < LimLow THEN
	Y_gaintrack := LimLow - Y;	
	Y := LimLow;
ELSIF Y > LimHigh THEN
	Y_gaintrack := LimHigh - Y;
	Y := LimHigh;
ELSE		
	Y_gaintrack := 0;
END_IF


(*
fse 17.10.2023:
- adjust anti-windup according to AixLib implementation

pos 23.10.2020:
- no anti-wind up on reset
- possibility to provide an offset value for Y

aku 24.09.2019: 
- first implementation
*)

END_FUNCTION_BLOCK

// ---- oscat_basic/POUs/Engineering/Control/FB_Integrate.TcPOU
FUNCTION_BLOCK FB_Integrate
VAR_INPUT
	run : BOOL 	:= TRUE;	// Set true for running integration
	in 	: REAL;				// integrated value
	K 	: REAL 	:= 1.0;		// factor
	RST	: BOOL  :=FALSE;	// set true for reinitialization
	inStart : REAL :=0; 		// start value
END_VAR

VAR_OUTPUT
	out 	: REAL;
END_VAR

VAR
	in_last : REAL;
	init: BOOL;
	last: TIME;
	tx: TIME;
END_VAR

(*read system time *)
tx := TIME();

//reset integration
IF RST = TRUE THEN
	init := FALSE;	
	out := inStart;
END_IF

IF NOT init THEN	//init last_in and skip integration for the first run
	init := TRUE;
	in_last := in;
	out := inStart;
ELSIF run THEN
	out := (in + in_last) * 0.5E-3 * TIME_TO_REAL(tx-last) * K + out;	//integration with trapezoidal rule
	in_last := in;
END_IF;
last := tx;	//save last time

END_FUNCTION_BLOCK

// ---- oscat_basic/POUs/Engineering/signal processing/FB_OutLinear.TcPOU
FUNCTION_BLOCK FB_OutLinear
VAR
	//Properties
	bError 				: BOOL 				:= FALSE;
	stIOConv			: IO_TERMINAL_PARAMETERS;
	
	//value
	fValueOut			: REAL;
	
	//Raw value
	nValueOutRaw		AT %Q* : INT;
END_VAR

PROPERTY Error : BOOL
GET
Error := THIS^.bError;
END_GET
SET
THIS^.bError := Error;
END_SET
END_PROPERTY

PROPERTY IO_Conversion : REFERENCE TO IO_TERMINAL_PARAMETERS
GET
IO_Conversion REF= THIS^.stIOConv;
END_GET
SET
THIS^.stIOConv := IO_Conversion;
END_SET
END_PROPERTY

PROPERTY ValueOut : REAL
GET
ValueOut := THIS^.fValueOut;
END_GET
SET
THIS^.fValueOut := ValueOut;
END_SET
END_PROPERTY

METHOD Write
nValueOutRaw := REAL_TO_INT(F_LIN2(X:=fValueOut,X1:=stIOConv.cValue1,Y1:=stIOConv.cValue1Raw,X2:=stIOConv.cValue2,Y2:=stIOConv.cValue2Raw));
END_METHOD

END_FUNCTION_BLOCK

// ---- oscat_basic/POUs/Engineering/Control/FT_IMP.TcPOU
FUNCTION_BLOCK FT_IMP
VAR_INPUT
	in : REAL;
	T : TIME;
	K : REAL := 1.0;
END_VAR
VAR_OUTPUT
	out : REAL;
END_VAR
VAR
	t1 : FT_PT1;
END_VAR

(*
version 1.1	3 Jan 2007
programmer 	hugo
tested by	oscat

FT_IMP is 	an impulse filter (high pass filter) with the time T and factor K.
 
*)

T1(in:= in, T:=T);
out := (in - t1.out) * K;

(*
hm 3.1.2007	rev 1.1
	added factor K

*)

END_FUNCTION_BLOCK

// ---- oscat_basic/POUs/Engineering/Control/FT_PI.TcPOU
FUNCTION_BLOCK FT_PI
VAR_INPUT
	IN : REAL;
	KP : REAL := 1.0;
	KI : REAL := 1.0;
	ILIM_L : REAL := -1E38;
	ILIM_H : REAL := 1E38;
	IEN : BOOL := TRUE;
	RST : BOOL;
END_VAR
VAR_OUTPUT
	Y : REAL;
	LIM : BOOL;
END_VAR
VAR
	integ : FT_INT;
END_VAR

(*
version 2.0	3. jun 2008
programmer 	hugo
tested by		tobias

FT_PI is a PI controller.
The PID controller works according to the fomula Y = IN *(KP+ KI * INTEG(e) ).
a rst will reset the integrator to 0
ilim_h and iLim_l set the possible output range of the internal integrator.
the output flags lim will signal that the output limits are active.

default values for KP = 1, KI = 1, ILIM_L = -1E37, iLIM_H = +1E38.
*)

(* run integrator *)
integ(IN := IN, K := KI, RUN := IEN, RST := RST, OUT_MIN := ILIM_L, OUT_MAX := ILIM_H);

(* check if integrator has reached its limits and set overflow *)
LIM := integ.LIM;
Y := KP * IN + integ.Out;



(* revision history
hm 	3. jun. 2008 	rev 2.0
	original version


*)

END_FUNCTION_BLOCK

// ---- oscat_basic/POUs/Engineering/Control/FT_PID.TcPOU
FUNCTION_BLOCK FT_PID
VAR_INPUT
	IN : REAL;
	KP : REAL := 1.0;
	TN : REAL := 1.0;
	TV : REAL := 1.0;
	ILIM_L : REAL := -1.0E38;
	ILIM_H : REAL := 1.0E38;
	IEN : BOOL := TRUE;
	RST : BOOL;
END_VAR
VAR_OUTPUT
	Y : REAL;
	LIM : BOOL;
END_VAR
VAR
	integ : FT_INT;
	diff : FT_DERIV;
END_VAR

(*
version 2.1	11. mar. 2009
programmer 	hugo
tested by		tobias

FT_PI is a PI controller.
The PID controller works according to the fomula Y = IN *(KP+ KI * INTEG(e) ).
a rst will reset the integrator to 0
ilim_h and iLim_l set the possible output range of the internal integrator.
the output flags lim will signal that the output limits are active.

default values for KP = 1, KI = 1, ILIM_L = -1E37, iLIM_H = +1E38.
*)

(* run integrator only if TN > 0 *)
IF TN > 0.0 THEN
	integ(IN := IN, K := 1.0 / TN, RUN := IEN, RST := RST, OUT_MIN := ILIM_L, OUT_MAX := ILIM_H);
ELSE
	integ(RST := TRUE);
END_IF;

(* run differentiator *)
diff(IN := IN, K := TV);

(* combine both values *)
Y := KP * (integ.Out + diff.out + IN);

(* check if integrator has reached its limits and set overflow *)
LIM := integ.LIM;



(* revision history
hm 3. jun. 2008 	rev 2.0
	original version

hm	11. mar. 2009	rev 2.1
	real constants updated to new systax using dot

*)

END_FUNCTION_BLOCK

// ---- oscat_basic/POUs/Engineering/Control/FT_PIW.TcPOU
FUNCTION_BLOCK FT_PIW
VAR_INPUT
	IN : REAL;
	KP : REAL := 1.0;
	KI : REAL := 1.0;
	LIM_L : REAL := -1E38;
	LIM_H : REAL := 1E38;
	RST : BOOL;
END_VAR
VAR_OUTPUT
	Y : REAL;
	LIM : BOOL;
END_VAR
VAR
	integ : FT_INT;
END_VAR

(*
version 1.0	3. jun 2008
programmer 	hugo
tested by		tobias

FT_PIW is a PI controller.
The PID controller works according to the fomula Y = IN *(KP+ KI * INTEG(e) ).
a rst will reset the integrator to 0
ilim_h and iLim_l set the possible output range of the internal integrator.
the output flag lim will signal that the output limits are active.
the controller is equipped with anti wind_up circuitry that stops the integrator when lim_h or lim_l is reached


default values for KP = 1, KI = 1, ILIM_L = -1E37, iLIM_H = +1E38.
*)

(* run integrator *)
integ(IN := IN, K := KI, RUN := NOT LIM, RST := RST);

(* set output value *)
Y := KP * IN + integ.Out;

(* check for limits and set integrator for anti wind up *)
IF Y < LIM_L THEN
	Y := LIM_L;
	LIM := TRUE;
ELSIF Y > LIM_H THEN
	Y := LIM_H;
	LIM := TRUE;
ELSE
	LIM := FALSE;
END_IF;



(* revision history
hm 	3. jun. 2008 	rev 1.0
	original version


*)

END_FUNCTION_BLOCK

// ---- oscat_basic/POUs/Engineering/Control/FT_TN16.TcPOU
FUNCTION_BLOCK FT_TN16
VAR_INPUT
	in : REAL;
	T : TIME;
END_VAR
VAR_OUTPUT
	out : REAL;
	trig : BOOL;
END_VAR
VAR
	length : INT := 16;
	X : ARRAY[0..15] OF REAL;
	cnt : INT;
	last : TIME;
	tx: TIME;
	init: BOOL;
END_VAR

(*
version 1.1	16 sep 2007
programmer 	hugo
tested by		tobias

FT_TN16 is delay function, it will delay a signal by a specified time : T and will store 16 values of in before they are put thru to out.
for higher or lower resolution please use FT_TN8 or FT_TN64 instead.
 
*)

(* read system time *)
tx := DWORD_TO_TIME(T_PLC_MS());

trig := FALSE;
IF NOT init THEN
	x[cnt] := in;
	init := TRUE;
	last := tx;
ELSIF tx - last >= T / length THEN
	IF cnt = length - 1 THEN cnt := 0; ELSE cnt := cnt + 1; END_IF;
	Out := X[cnt];
	x[cnt] := in;
	last := tx;
	Trig := TRUE;
END_IF;

(* revision history
hm		1. jan 2007	rev 1.0
	original version

hm		16. sep 2007	rev 1.1
	changes time() to T_plc_ms() for compatibility reasons

*)

END_FUNCTION_BLOCK

// ---- oscat_basic/POUs/Engineering/Control/FT_TN64.TcPOU
FUNCTION_BLOCK FT_TN64
VAR_INPUT
	in : REAL;
	T : TIME;
END_VAR
VAR_OUTPUT
	out : REAL;
	trig: BOOL;
END_VAR
VAR
	length : INT := 64;
	X : ARRAY[0..63] OF REAL;
	cnt : INT;
	last : TIME;
	tx: TIME;
	init: BOOL;
END_VAR

(*
version 1.1	15 sep 2007
programmer 	hugo
tested by		tobias

FT_TN7 is delay function, it will delay a signal by a specified time : T and will store 64 values of in before they are put thru to out.
if lower resolution is needed, pls use FT_TN8 or FT_TN16 instead.
 
*)

(* read system time *)
tx := DWORD_TO_TIME(T_PLC_MS());

trig := FALSE;
IF NOT init THEN
	x[cnt] := in;
	init := TRUE;
	last := tx;
ELSIF tx - last >= T / length THEN
	IF cnt = length - 1 THEN cnt := 0; ELSE cnt := cnt + 1; END_IF;
	Out := X[cnt];
	x[cnt] := in;
	last := tx;
	trig := TRUE;
END_IF;

(* revision history
hm		1. jan 2007		rev 1.0
	original version

hm		16. sep 2007	rev 1.1
	changes time() to T_plc_ms() for compatibility reasons

*)

END_FUNCTION_BLOCK

// ---- oscat_basic/POUs/Engineering/Control/FT_TN8.TcPOU
FUNCTION_BLOCK FT_TN8
VAR_INPUT
	in : REAL;
	T : TIME;
END_VAR
VAR_OUTPUT
	out : REAL;
	trig: BOOL;
END_VAR
VAR
	length : INT := 8;
	X : ARRAY[0..7] OF REAL;
	cnt : INT;
	last : TIME;
	tx: TIME;
	init: BOOL;
END_VAR

(*
version 1.1	15 Sep 2007
programmer 	hugo
tested by		tobias

FT_TN8 is delay function, it will delay a signal by a specified time : T and will store 8 values of in before they are put thru to out.
if higher resolution is needed, pls use FT_TN16 or FT_TN64 instead.
 
*)

tx := DWORD_TO_TIME(T_PLC_MS());
trig := FALSE;
IF NOT init THEN
	x[cnt] := in;
	init := TRUE;
	last := tx;
ELSIF tx - last >= T / length THEN
	IF cnt = length - 1 THEN cnt := 0; ELSE cnt := cnt + 1; END_IF;
	Out := X[cnt];
	x[cnt] := in;
	last := tx;
	trig := TRUE;
END_IF;

(* revision history
hm		1. jan 2007		rev 1.0
	original version

hm		16. sep 2007	rev 1.1
	changes time() to T_plc_ms() for compatibility reasons

*)

END_FUNCTION_BLOCK

// ---- oscat_basic/POUs/Engineering/Control/HYST.TcPOU
FUNCTION_BLOCK HYST
VAR_INPUT
	In : REAL;
	ON : REAL;
	OFF : REAL;
END_VAR
VAR_OUTPUT
	Q : BOOL;
	win : BOOL;
END_VAR


(*
version 1.0	2. jun. 2008
programmer 	hugo
tested BY	oscat

This Hystereses function has two modes:
1. if on > off then Q will be switched high when in > on and switched low when in < off.
2. if on < off then Q will be switched high when in < on and switched low when in > off.
the output win will be high when in is between low and high.

*)

IF ON >= OFF THEN
	IF IN < OFF THEN
		Q := FALSE;
		WIN := FALSE;
	ELSIF  IN > ON THEN
		Q := TRUE;
		WIN := FALSE;
	ELSE
		WIN := TRUE;
	END_IF;
ELSE
	IF IN > OFF THEN
		Q := FALSE;
		WIN := FALSE;
	ELSIF  IN < ON THEN
		Q := TRUE;
		WIN := FALSE;
	ELSE
		WIN := TRUE;
	END_IF;
END_IF;


(* revision history
hm		2.  jun 2008	rev 1.0
	original version

*)

END_FUNCTION_BLOCK

// ---- oscat_basic/POUs/Engineering/Control/HYST_1.TcPOU
FUNCTION_BLOCK HYST_1
VAR_INPUT
	In : REAL;
	high : REAL;
	low : REAL;
END_VAR
VAR_OUTPUT
	Q : BOOL;
	win : BOOL;
END_VAR


(*
version 1.1	2. jun. 2008
programmer 	hugo
tested BY	oscat

this hysteresis function switches the output high if the input signal reaches obove high and will switch to low when the input falls back below low value.
a separate output mid is set if the input stays between low and high value.

*)

IF in < low THEN
	Q := FALSE;
	win := FALSE;
ELSIF in > high THEN
	Q := TRUE;
	win := FALSE;
ELSE
	win := TRUE;
END_IF;




(* revision history
hm		4.  aug. 2006	rev 1.0
	original version

hm		2. jun. 2008	rev 1.1
	improved performance
*)

END_FUNCTION_BLOCK

// ---- oscat_basic/POUs/Engineering/Control/HYST_2.TcPOU
FUNCTION_BLOCK HYST_2
VAR_INPUT
	IN : REAL;
	VAL : REAL;
	HYS : REAL;
END_VAR
VAR_OUTPUT
	Q : BOOL;
	WIN: BOOL;
END_VAR
VAR
	tmp: REAL;
END_VAR


(*
version 1.2	2. jun. 2008
programmer 	oscat
tested BY	oscat

this hysteresis function switches the output high if the input signal reaches obove val + hys/2 and will switch to low when the input falls back below val - hys/2 value.
a separate output mid is set if the input stays between low and high value.

*)

tmp := val - hys * 0.5;
IF in < tmp THEN
	Q := FALSE;
	win := FALSE;
ELSIF in > tmp + hys THEN
	Q := TRUE;
	win := FALSE;
ELSE
	win := TRUE;
END_IF;



(* revision history
hm		4. aug 2006	rev 1.0
	original version

hm		5. jan 2008	rev 1.1
	improved code for better performance

hm		2. jun. 2008	rev 1.2
	improved performance
*)

END_FUNCTION_BLOCK

// ---- oscat_basic/POUs/Engineering/Control/HYST_3.TcPOU
FUNCTION_BLOCK HYST_3
VAR_INPUT
	in : REAL;
	hyst : REAL;
	val1 : REAL;
	val2 : REAL;
END_VAR
VAR_OUTPUT
	Q1 : BOOL;
	Q2 : BOOL;
END_VAR
VAR
	X: REAL;
END_VAR

(*
version 1.2	5 jan 2008
programmer 	oscat
tested BY	oscat

this is a double hysteresis function. Out1 follows a hysteresis function defined by val1and hyst, while out 2 follows val2 and hyst.
if the input signal is between the two hysteresis switches (val1 and val2) then non of the outputs is active.

*)

X := hyst * 0.5;
IF in < val1 - X THEN
	q1 := TRUE;
ELSIF in > val1 + X THEN
	q1 := FALSE;
END_IF;
IF in < val2 - X THEN
	q2 := FALSE;
ELSIF in > val2 + X THEN
	q2 := TRUE;
END_IF;



(* revision history
hm	22. jan 2007	rev 1.0
	original version

hm	27. dec 2007	rev 1.1
	changed code for better performance

hm	5. jan 2008	rev 1.2
	further performance iprovements

*)

END_FUNCTION_BLOCK

// ---- oscat_basic/POUs/Engineering/Conversion/C_TO_F.TcPOU
FUNCTION C_TO_F : REAL
VAR_INPUT
	celsius : REAL;
END_VAR


(*
version 1.1	11. mar. 2009
programmer 	hugo
tested by		tobias

this function converts celsius  to fahrenheit 

*)

C_TO_F := celsius * 1.8 + 32.0;


(* revision history

hm	4. aug. 2006	rev 1.0
	original version

hm	11. mar. 2009	rev 1.1
	real constants updated to new systax using dot

*)

END_FUNCTION

// ---- oscat_basic/POUs/Engineering/Conversion/C_TO_K.TcPOU
FUNCTION C_TO_K : REAL
VAR_INPUT
	Celsius : REAL;
END_VAR


(*
version 1.1	19. aug 2009
programmer 	hugo
tested by		tobias

this function converts celsius to kelvin
*)

C_TO_K := Celsius - phys.T0;

(* revision history

hm	4. aug 2006	rev 1.0
	original version

hm	19. aug 2009	rev 1.1
	fixed calculation error

*)

END_FUNCTION

// ---- oscat_basic/POUs/Engineering/Conversion/DEG_TO_DIR.TcPOU
FUNCTION DEG_TO_DIR : STRING(3)
VAR_INPUT
	DEG : INT;
	N : INT;
	L : INT;
END_VAR
VAR
	ly: INT;
END_VAR


(*
version 1.1	22. oct. 2008
programmer 	hugo
tested by		oscat

this function converts degrees in compass direction.
the function supports output in english (L=0) and german (L=1).

*)

IF L = 0 THEN ly := LANGUAGE.DEFAULT; ELSE ly := MIN(L, LANGUAGE.LMAX); END_IF;
DEG_TO_DIR := LANGUAGE.DIRS[ly, ((SHL(DEG,N-1) + 45) / 90) MOD SHL(INT#2,N)*SHR(INT#8,N)];



(*
DIR := ((SHL(DEG,N-1) + 45) / 90) MOD SHL(INT#2,N);
explanation :
DIR is calculated BY the following formula:
DIR := ((DIR + 45) / 90) MOD 4 if N = 1 digit
North = 0, East = 1 ....
DIR := ((DIR + 22,5) / 45) MOD 8 if N = 2 digit
convert to integer calculation
DIR := ((DIR*2 + 45) / 90) MOD 8
N = 0, NE = 1 ....
ther above formula replaces 2^N with shift for performance
*)



(* revision histroy
hm	11. jun. 2008	rev 1.0
	original release

hm	22. oct. 2008	rev 1.1
	changed size of string variables to 30
*)

END_FUNCTION

// ---- oscat_basic/POUs/Engineering/Conversion/ENERGY.TcPOU
FUNCTION_BLOCK ENERGY
VAR_INPUT
	J : REAL;
	C : REAL;
	Wh : REAL;
END_VAR
VAR_OUTPUT
	YJ : REAL;
	YC : REAL;
	YWh : REAL;
END_VAR


(*
version 1.2	16. jan. 2010
programmer 	hugo
tested by		oscat

this function converts different energy units
any unused input can simply be left open.
different inputs connected at the same time will be added up.
*)

YJ := J + Wh * 3600.0 + C * 4.1868;
YC := YJ * 0.238845896627496;
YWh := YJ * 2.7777777778E-004;

(*
Arbeit, Energie, Joule* J 1 J = 1 N · m = 1 W · s = (1/3,6) E–6 kW · h = 1 kg · m2/s2
Wärmemenge Kilowattstunde kW · h 1 kW · h = 3,6 MJ = 860 kcal
Elektronvolt eV 1 eV = 160,218 92 E–21 J
Erg erg 1 erg = 1E–7 J
Kalorie calorie 1 calalorie = 4,1868 J = 1,163 E–3 W · h
Therm therm 1 therm = 105,50 · 106 J
*)

(* revision history

hm	27. mar. 2007	rev 1.0
	original version

hm	11. mar. 2009	rev 1.1
	improved code

hm 16. jan 2010	rev 1.2
	avoid the string cal in comments for codesys import bug


*)

END_FUNCTION_BLOCK

// ---- oscat_basic/POUs/Engineering/Conversion/F_TO_PT.TcPOU
FUNCTION F_TO_PT : TIME
VAR_INPUT
	F : REAL;
END_VAR


(*
version 1.1	11. mar. 2009
programmer 	hugo
tested by		tobias

this function converts frequency to periode time  
*)

F_TO_PT := DWORD_TO_TIME(REAL_TO_DWORD(1.0 / F * 1000.0));


(* revision history

hm	4. aug. 2006	rev 1.0
	original version

hm	11. mar. 2009	rev 1.1
	real constants updated to new systax using dot

*)

END_FUNCTION

// ---- oscat_basic/POUs/Engineering/Conversion/KMH_TO_MS.TcPOU
FUNCTION KMH_TO_MS : REAL
VAR_INPUT
	kmh : REAL;
END_VAR


(*
version 1.1	6 jan 2007
programmer 	hugo
tested by		tobias

this function converts velocities from Kilometers / hour to Meters / Second

*)

KMH_TO_MS := kmh * 0.2777777777777;

(* revision history
hm	4. feb 2007		rev 1.0
	original version

hm	6. jan 2008		rev 1.1
	improved performance

*)

END_FUNCTION

// ---- oscat_basic/POUs/Engineering/Conversion/MS_TO_KMH.TcPOU
FUNCTION MS_TO_KMH : REAL
VAR_INPUT
	ms : REAL;
END_VAR


(*
version 1.0	4 Feb 2007
programmer 	hugo
tested by		tobias

this function converts velocities from Meters / Second to Kilometers / hour.

*)

MS_TO_KMH := ms * 3.6;

END_FUNCTION

// ---- oscat_basic/POUs/Engineering/measurements/CALIBRATE.TcPOU
FUNCTION_BLOCK CALIBRATE
VAR_INPUT
	X : REAL;
	CO : BOOL;
	CS : BOOL;
END_VAR
VAR_INPUT CONSTANT
	Y_Offset : REAL;
	Y_Scale : REAL;
END_VAR
VAR_OUTPUT
	Y : REAL;
END_VAR
VAR RETAIN
	offset : REAL;
	Scale : REAL := 1.0;
END_VAR

(*
	version 1.3	11. mar. 2009
	programmer 	hugo
	tested BY		hans

Calibrate allows for offset and scale calibration of an analog input.
offset is calibrated to a stored reference Y_offset while CO is true.
after the offset is calibrated, scale can be calibrated to a reference value Y_scale while CS is true.
*)

(* check for calibration *)
IF CO THEN
	OFFSET := Y_Offset - X;
ELSIF CS THEN
	SCALE := Y_scale / (X + OFFSET);
END_IF;
(* calculate output *)
Y := (X + OFFSET) * SCALE;


(* revision history
hm 22.2.2007		rev 1.2
	changed VAR RETAIN PERSISTENT to VAR RETAIN for better compatibility
	wago lon contollers do not support persisitent

hm	11. mar. 2009	rev 1.3
	changed real constants to use dot syntax

*)

END_FUNCTION_BLOCK

// ---- oscat_basic/POUs/Engineering/measurements/FLOW_METER.TcPOU
FUNCTION_BLOCK FLOW_METER
VAR_INPUT
	VX : REAL;
	E : BOOL;
	RST : BOOL;
END_VAR
VAR_INPUT CONSTANT
	PULSE_MODE : BOOL;
	UPDATE_TIME : TIME := t#1s;
END_VAR
VAR_OUTPUT
	F : REAL;
END_VAR
VAR_IN_OUT
	X : REAL;
	Y : UDINT;
END_VAR
VAR
	tx, tl : TIME;
	int1 : INTEGRATE;
	init: BOOL;
	e_last : BOOL;
	tmp: INT;
	x_last : REAL;
	y_last : UDINT;
END_VAR

(*
version 1.0	23. jan. 2011
programmer 	hugo
tested by	oscat

Flow meter measures flow according to gated time or pulses.

*)

IF NOT init THEN	(* init on power up *)
	init := TRUE;
	tl := tx;
	x_last := X;
	y_last := Y;
	int1.K := 2.7777777777777777E-4;
END_IF;

(* run integrator *)
int1(E := NOT (RST OR PULSE_MODE) AND E, X := VX, Y := X);	(* gated operation *)

IF RST THEN		(* reset *)
	X := 0.0;
	Y := 0;
	tl := tx;
	x_last := 0.0;
	y_last := 0;
ELSIF E AND PULSE_MODE THEN	(* check for pulse mode *)
	IF NOT e_last THEN X := X + VX; END_IF;
END_IF;
e_last := E;

(* reduce X to be less than 1 and increase Y respectively *)
IF X > 1.0 THEN
	tmp := FLOOR(X);
	Y := Y + INT_TO_UDINT(tmp);
	X := X - INT_TO_REAL(tmp);
END_IF;

(* calculate the current flow *)
tx := DWORD_TO_TIME(T_PLC_MS());
IF tx - tl >= UPDATE_TIME AND UPDATE_TIME > t#0s THEN
	F := (UDINT_TO_REAL(Y - y_last) + X - x_last) / TIME_TO_REAL(tx - tl) * 3.6E6;
	y_last := Y;
	x_last := X;
	tl := tx;
END_IF;



(* revision history
hm	23. jan. 2011	rev 1.0
	original version

*)

END_FUNCTION_BLOCK

// ---- oscat_basic/POUs/Engineering/measurements/METER_STAT.TcPOU
FUNCTION_BLOCK METER_STAT
VAR_INPUT
	IN : REAL;
	DI : DATE;
	RST : BOOL;
END_VAR
VAR_IN_OUT
	Last_Day : REAL;
	Current_Day : REAL;
	Last_Week : REAL;
	Current_Week : REAL;
	Last_Month : REAL;
	Current_Month : REAL;
	Last_Year : REAL;
	Current_Year : REAL;
END_VAR
VAR RETAIN
	Year_Start : REAL;
	Month_Start : REAL;
	Week_Start : REAL;
	Day_Start : REAL;
	last_run: DATE;
END_VAR

(*
	version 1.3	18. jul. 2009
	programmer 	oscat
	tested BY		oscat

METER_STAT runs statistics of a metered value, it calculates the current week, day, month and year consumption and stores the corresponding last day, week, month and year value.

*)

IF rst THEN
	Last_Day := 0.0;
	Current_Day := 0.0;
	Day_start := IN;
	Last_week := 0.0;
	Current_week := 0.0;
	Week_start := in;
	Last_month := 0.0;
	Current_month := 0.0;
	month_start := in;
	last_year := 0.0;
	current_year := 0.0;
	year_start := in;
ELSE
	Current_Day := IN - Day_Start;
	Current_Week := In - Week_Start;
	Current_Month := IN - Month_Start;
	Current_Year := IN - Year_Start;
END_IF;

